KUKA KRL program: EPS_2_25694_SR01_A_20251117072407.src

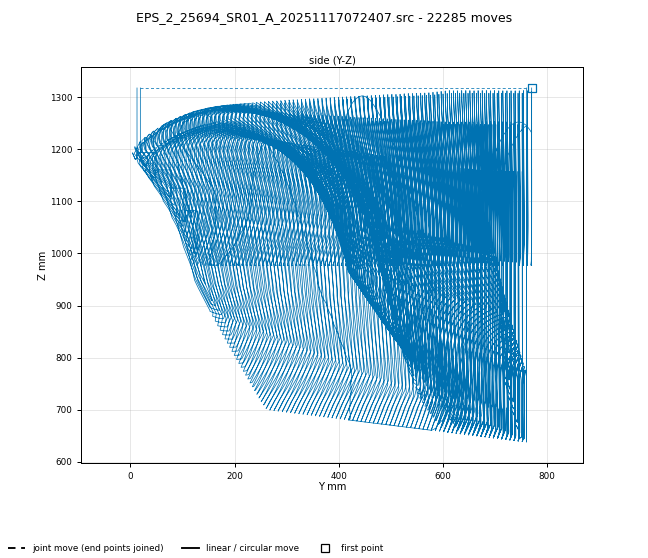
[picture p0: tool path of EPS_2_25694_SR01_A_20251117072407.src, 22285 of 22287 moves have a stored position in this frame; points joined in program order, loops and branches not executed]
&ACCESS RVP
&REL 4
&COMMENT QRS 19112012
&PARAM EDITMASK = *
DEF PART()
EXT BAS (BAS_COMMAND :IN,REAL :IN )
INT I
BAS (#INITMOV,0 )

;KUKA QRS Post kuka4.cps  Date:22-06-2017 !

File_ID=2905

QRS_PRE_INIT()

;Init var - Until changes are made in qrs_pre_init
Outlet_Square_prg=0
Inlet_1_Square_prg=0
Inlet_2_Square_prg=0
Inlet_3_Square_prg=0
Inlet_4_Square_prg=0
Inlet_5_Square_prg=0

Outlet_1={X 0.000, Y 612.000, Z 1041.000, B 0.000, E1 0.000 }
Inlet_1={X 0.000, Y 612.000, Z 981.000, B 0.000, E1 90.000 }
Inlet_2={X 0.000, Y 687.170, Z 452.000, B 0.000, E1 260.000 }
Outlet_1_type=533
Inlet_1_type=533
Inlet_2_type=251
;QRS#1=Sidecore dimensions
;QRS#2=525-21" Concrete
;QRS#3=525-21" Concrete
;QRS#4=250-10" PVC SDR 35
;QRS#5=
;QRS#6=
;QRS#7=
;QRS#8=
;QRS#9=S306-32
;QRS#10=S306-32
;QRS#11=14M PSX
;QRS#12=
;QRS#13=
;QRS#14=
;QRS#15=
;QRS#16=1524x152x1753 5,75'
;QRS#17=EPS Height
;QRS#18=1307,5
;QRS#19=*
;QRS#20= UPDATED VERSION 22-06-2017
;QRS#21=*
Outlet_Square=0350
Inlet_1_Square=0350
Inlet_2_Square=0100
Inlet_3_Square=0
Inlet_4_Square=0
Inlet_5_Square=0
Mill_Square=1
Outlet_Square_Prg=263
Inlet_1_Square_prg=263
Inlet_2_Square_prg=205

QRS_INIT()

$ADVANCE=5

; T1
PTP {E1 171.718,E2 171.718}
PTP {X 0,Y 770.023,A -85,B 0,C 180,E1 171.718,E2 171.718,E3 0,E4 0,E5 0,E6 0}
QRS_SPEED_INIT()
LIN {X 0,Y 770.023,Z 1317.5,A -85,B 0,C 180,E1 171.718,E2 171.718,E3 0,E4 0,E5 0,E6 0} C_VEL
LIN {X 0,Y 770.023,Z 1241.436,A -85,B 0,C 180,E1 171.718,E2 171.718} C_VEL
LIN {X 0,Y 770.023,Z 1233.323,A -85,B 0,C 180,E1 171.718,E2 171.718} C_VEL
LIN {X 0,Y 769.973,Z 1231.44,A -85,B 0,C 180,E1 171.917,E2 171.917} C_VEL
LIN {X 0,Y 769.865,Z 1236.016,A -85,B 0,C 180,E1 172.868,E2 172.868} C_VEL
LIN {X 0,Y 769.858,Z 1240.057,A -85,B 0,C 180,E1 173.85,E2 173.85} C_VEL
LIN {X 0,Y 769.972,Z 1243.895,A -85,B 0,C 180,E1 174.972,E2 174.972} C_VEL
LIN {X 0,Y 769.797,Z 1246.945,A -85,B 0,C 180,E1 176.09,E2 176.09} C_VEL
LIN {X 0,Y 769.867,Z 1249.135,A -85,B 0,C 180,E1 177.209,E2 177.209} C_VEL
LIN {X 0,Y 769.978,Z 1250.214,A -85,B 0,C 180,E1 177.954,E2 177.954} C_VEL
LIN {X 0,Y 769.814,Z 1251.211,A -85,B 0,C 180,E1 179.07,E2 179.07} C_VEL
LIN {X 0,Y 769.987,Z 1251.132,A -85,B 0,C 180,E1 180.93,E2 180.93} C_VEL
LIN {X 0,Y 769.924,Z 1250.495,A -85,B 0,C 180,E1 181.674,E2 181.674} C_VEL
LIN {X 0,Y 769.997,Z 1248.968,A -85,B 0,C 180,E1 182.791,E2 182.791} C_VEL
LIN {X 0,Y 769.853,Z 1246.736,A -85,B 0,C 180,E1 183.909,E2 183.909} C_VEL
LIN {X 0,Y 769.92,Z 1243.606,A -85,B 0,C 180,E1 185.028,E2 185.028} C_VEL
LIN {X 0,Y 769.995,Z 1241.081,A -85,B 0,C 180,E1 185.775,E2 185.775} C_VEL
LIN {X 0,Y 769.852,Z 1237.005,A -85,B 0,C 180,E1 186.824,E2 186.824} C_VEL
LIN {X 0,Y 769.887,Z 1232.516,A -85,B 0,C 180,E1 187.791,E2 187.791} C_VEL
LIN {X 0,Y 769.947,Z 1226.703,A -85,B 0,C 180,E1 188.87,E2 188.87} C_VEL
LIN {X 0,Y 769.873,Z 1220.945,A -85,B 0,C 180,E1 189.814,E2 189.814} C_VEL
LIN {X 0,Y 769.962,Z 1214.413,A -85,B 0,C 180,E1 190.758,E2 190.758} C_VEL
LIN {X 0,Y 769.919,Z 1207.115,A -85,B 0,C 180,E1 191.706,E2 191.706} C_VEL
LIN {X 0,Y 769.869,Z 1200.05,A -85,B 0,C 180,E1 192.54,E2 192.54} C_VEL
LIN {X 0,Y 769.952,Z 1192.23,A -85,B 0,C 180,E1 193.373,E2 193.373} C_VEL
LIN {X 0,Y 769.972,Z 1184.939,A -85,B 0,C 180,E1 194.091,E2 194.091} C_VEL
LIN {X 0,Y 769.933,Z 1175.825,A -85,B 0,C 180,E1 194.91,E2 194.91} C_VEL
LIN {X 0,Y 769.965,Z 1167.286,A -85,B 0,C 180,E1 195.613,E2 195.613} C_VEL
LIN {X 0,Y 769.992,Z 1158.209,A -85,B 0,C 180,E1 196.301,E2 196.301} C_VEL
LIN {X 0,Y 769.94,Z 1148.195,A -85,B 0,C 180,E1 196.999,E2 196.999} C_VEL
LIN {X 0,Y 769.971,Z 1137.702,A -85,B 0,C 180,E1 197.665,E2 197.665} C_VEL
LIN {X 0,Y 769.976,Z 1127.341,A -85,B 0,C 180,E1 198.267,E2 198.267} C_VEL
LIN {X 0,Y 769.983,Z 1116.994,A -85,B 0,C 180,E1 198.819,E2 198.819} C_VEL
LIN {X 0,Y 769.976,Z 1105.571,A -85,B 0,C 180,E1 199.373,E2 199.373} C_VEL
LIN {X 0,Y 769.917,Z 1094.356,A -85,B 0,C 180,E1 199.868,E2 199.868} C_VEL
LIN {X 0,Y 769.976,Z 1080.704,A -85,B 0,C 180,E1 200.4,E2 200.4} C_VEL
LIN {X 0,Y 769.957,Z 1068.91,A -85,B 0,C 180,E1 200.812,E2 200.812} C_VEL
LIN {X 0,Y 769.908,Z 1058.029,A -85,B 0,C 180,E1 201.153,E2 201.153} C_VEL
LIN {X 0,Y 769.994,Z 1042.62,A -85,B 0,C 180,E1 201.561,E2 201.561} C_VEL
LIN {X 0,Y 769.955,Z 1029.278,A -85,B 0,C 180,E1 201.861,E2 201.861} C_VEL
LIN {X 0,Y 769.84,Z 1017.832,A -85,B 0,C 180,E1 202.082,E2 202.082} C_VEL
LIN {X 0,Y 769.939,Z 1002.652,A -85,B 0,C 180,E1 202.304,E2 202.304} C_VEL
LIN {X 0,Y 769.825,Z 984.624,A -85,B 0,C 180,E1 202.504,E2 202.504} C_VEL
LIN {X 0,Y 769.657,Z 979.091,A -85,B 0,C 180,E1 202.564,E2 202.564} C_VEL
LIN {X 0,Y 769.078,Z 977.53,A -85,B 0,C 180,E1 202.604,E2 202.604} C_VEL
LIN {X 0,Y 770.082,Z 977.53,A -85,B 0,C 180,E1 202.974,E2 202.974} C_VEL
LIN {X 0,Y 769.685,Z 977.53,A -85,B 0,C 180,E1 203.948,E2 203.948} C_VEL
LIN {X 0,Y 769.897,Z 977.53,A -85,B 0,C 180,E1 208.082,E2 208.082} C_VEL
LIN {X 0,Y 769.516,Z 977.53,A -85,B 0,C 180,E1 210.601,E2 210.601} C_VEL
LIN {X 0,Y 769.917,Z 977.53,A -85,B 0,C 180,E1 212.388,E2 212.388} C_VEL
LIN {X 0,Y 769.483,Z 977.53,A -85,B 0,C 180,E1 214.641,E2 214.641} C_VEL
LIN {X 0,Y 770.049,Z 977.53,A -85,B 0,C 180,E1 217.324,E2 217.324} C_VEL
LIN {X 0,Y 769.704,Z 977.53,A -85,B 0,C 180,E1 221.735,E2 221.735} C_VEL
LIN {X 0,Y 769.745,Z 977.53,A -85,B 0,C 180,E1 223.064,E2 223.064} C_VEL
LIN {X 0,Y 769.737,Z 977.53,A -85,B 0,C 180,E1 226.937,E2 226.937} C_VEL
LIN {X 0,Y 769.697,Z 977.53,A -85,B 0,C 180,E1 228.264,E2 228.264} C_VEL
LIN {X 0,Y 770.068,Z 977.53,A -85,B 0,C 180,E1 232.674,E2 232.674} C_VEL
LIN {X 0,Y 769.762,Z 977.53,A -85,B 0,C 180,E1 235.892,E2 235.892} C_VEL
LIN {X 0,Y 769.686,Z 977.53,A -85,B 0,C 180,E1 237.601,E2 237.601} C_VEL
LIN {X 0,Y 769.425,Z 977.53,A -85,B 0,C 180,E1 239.767,E2 239.767} C_VEL
LIN {X 0,Y 769.9,Z 977.53,A -85,B 0,C 180,E1 241.918,E2 241.918} C_VEL
LIN {X 0,Y 769.973,Z 977.53,A -85,B 0,C 180,E1 246.365,E2 246.365} C_VEL
LIN {X 0,Y 769.665,Z 977.53,A -85,B 0,C 180,E1 246.705,E2 246.705} C_VEL
LIN {X 0,Y 769.269,Z 977.53,A -85,B 0,C 180,E1 246.754,E2 246.754} C_VEL
LIN {X 0,Y 769.172,Z 977.768,A -85,B 0,C 180,E1 246.767,E2 246.767} C_VEL
LIN {X 0,Y 769.749,Z 993.425,A -85,B 0,C 180,E1 246.941,E2 246.941} C_VEL
LIN {X 0,Y 769.865,Z 1055.898,A -85,B 0,C 180,E1 247.57,E2 247.57} C_VEL
LIN {X 0,Y 769.803,Z 1068.07,A -85,B 0,C 180,E1 247.72,E2 247.72} C_VEL
LIN {X 0,Y 769.924,Z 1081.39,A -85,B 0,C 180,E1 247.941,E2 247.941} C_VEL
LIN {X 0,Y 769.888,Z 1094.597,A -85,B 0,C 180,E1 248.205,E2 248.205} C_VEL
LIN {X 0,Y 769.945,Z 1107.084,A -85,B 0,C 180,E1 248.505,E2 248.505} C_VEL
LIN {X 0,Y 769.959,Z 1120.713,A -85,B 0,C 180,E1 248.887,E2 248.887} C_VEL
LIN {X 0,Y 769.857,Z 1132.612,A -85,B 0,C 180,E1 249.265,E2 249.265} C_VEL
LIN {X 0,Y 769.961,Z 1143.963,A -85,B 0,C 180,E1 249.674,E2 249.674} C_VEL
LIN {X 0,Y 769.976,Z 1156.83,A -85,B 0,C 180,E1 250.195,E2 250.195} C_VEL
LIN {X 0,Y 769.92,Z 1169.12,A -85,B 0,C 180,E1 250.748,E2 250.748} C_VEL
LIN {X 0,Y 769.966,Z 1180.216,A -85,B 0,C 180,E1 251.303,E2 251.303} C_VEL
LIN {X 0,Y 769.976,Z 1191.366,A -85,B 0,C 180,E1 251.915,E2 251.915} C_VEL
LIN {X 0,Y 769.968,Z 1201.997,A -85,B 0,C 180,E1 252.556,E2 252.556} C_VEL
LIN {X 0,Y 769.956,Z 1212.08,A -85,B 0,C 180,E1 253.221,E2 253.221} C_VEL
LIN {X 0,Y 769.966,Z 1221.361,A -85,B 0,C 180,E1 253.887,E2 253.887} C_VEL
LIN {X 0,Y 769.995,Z 1229.576,A -85,B 0,C 180,E1 254.525,E2 254.525} C_VEL
LIN {X 0,Y 769.904,Z 1239.008,A -85,B 0,C 180,E1 255.323,E2 255.323} C_VEL
LIN {X 0,Y 769.901,Z 1246.661,A -85,B 0,C 180,E1 256.027,E2 256.027} C_VEL
LIN {X 0,Y 769.981,Z 1254.955,A -85,B 0,C 180,E1 256.865,E2 256.865} C_VEL
LIN {X 0,Y 769.899,Z 1262.523,A -85,B 0,C 180,E1 257.698,E2 257.698} C_VEL
LIN {X 0,Y 769.889,Z 1269.388,A -85,B 0,C 180,E1 258.53,E2 258.53} C_VEL
LIN {X 0,Y 769.994,Z 1276.399,A -85,B 0,C 180,E1 259.478,E2 259.478} C_VEL
LIN {X 0,Y 769.921,Z 1281.234,A -85,B 0,C 180,E1 260.186,E2 260.186} C_VEL
LIN {X 0,Y 769.846,Z 1286.993,A -85,B 0,C 180,E1 261.128,E2 261.128} C_VEL
LIN {X 0,Y 769.955,Z 1292.809,A -85,B 0,C 180,E1 262.232,E2 262.232} C_VEL
LIN {X 0,Y 769.885,Z 1297.298,A -85,B 0,C 180,E1 263.207,E2 263.207} C_VEL
LIN {X 0,Y 769.849,Z 1301.265,A -85,B 0,C 180,E1 264.223,E2 264.223} C_VEL
LIN {X 0,Y 769.951,Z 1303.746,A -85,B 0,C 180,E1 264.971,E2 264.971} C_VEL
LIN {X 0,Y 769.854,Z 1306.835,A -85,B 0,C 180,E1 266.09,E2 266.09} C_VEL
LIN {X 0,Y 769.819,Z 1309.08,A -85,B 0,C 180,E1 267.207,E2 267.207} C_VEL
LIN {X 0,Y 769.983,Z 1310.517,A -85,B 0,C 180,E1 268.325,E2 268.325} C_VEL
LIN {X 0,Y 769.856,Z 1311.187,A -85,B 0,C 180,E1 269.069,E2 269.069} C_VEL
LIN {X 0,Y 769.856,Z 1311.188,A -85,B 0,C 180,E1 270.929,E2 270.929} C_VEL
LIN {X 0,Y 769.923,Z 1310.164,A -85,B 0,C 180,E1 272.045,E2 272.045} C_VEL
LIN {X 0,Y 769.819,Z 1309.084,A -85,B 0,C 180,E1 272.79,E2 272.79} C_VEL
LIN {X 0,Y 769.853,Z 1306.84,A -85,B 0,C 180,E1 273.908,E2 273.908} C_VEL
LIN {X 0,Y 769.952,Z 1303.754,A -85,B 0,C 180,E1 275.027,E2 275.027} C_VEL
LIN {X 0,Y 769.844,Z 1299.884,A -85,B 0,C 180,E1 276.149,E2 276.149} C_VEL
LIN {X 0,Y 769.925,Z 1295.884,A -85,B 0,C 180,E1 277.111,E2 277.111} C_VEL
LIN {X 0,Y 769.924,Z 1291.346,A -85,B 0,C 180,E1 278.059,E2 278.059} C_VEL
LIN {X 0,Y 769.846,Z 1287.007,A -85,B 0,C 180,E1 278.87,E2 278.87} C_VEL
LIN {X 0,Y 769.921,Z 1281.25,A -85,B 0,C 180,E1 279.812,E2 279.812} C_VEL
LIN {X 0,Y 769.972,Z 1274.763,A -85,B 0,C 180,E1 280.756,E2 280.756} C_VEL
LIN {X 0,Y 769.879,Z 1267.512,A -85,B 0,C 180,E1 281.706,E2 281.706} C_VEL
LIN {X 0,Y 769.935,Z 1260.465,A -85,B 0,C 180,E1 282.537,E2 282.537} C_VEL
LIN {X 0,Y 769.965,Z 1252.697,A -85,B 0,C 180,E1 283.371,E2 283.371} C_VEL
LIN {X 0,Y 769.895,Z 1243.731,A -85,B 0,C 180,E1 284.248,E2 284.248} C_VEL
LIN {X 0,Y 769.951,Z 1236.134,A -85,B 0,C 180,E1 284.929,E2 284.929} C_VEL
LIN {X 0,Y 769.974,Z 1226.492,A -85,B 0,C 180,E1 285.719,E2 285.719} C_VEL
LIN {X 0,Y 769.941,Z 1217.541,A -85,B 0,C 180,E1 286.395,E2 286.395} C_VEL
LIN {X 0,Y 769.96,Z 1207.794,A -85,B 0,C 180,E1 287.069,E2 287.069} C_VEL
LIN {X 0,Y 769.966,Z 1198.499,A -85,B 0,C 180,E1 287.663,E2 287.663} C_VEL
LIN {X 0,Y 769.97,Z 1187.07,A -85,B 0,C 180,E1 288.327,E2 288.327} C_VEL
LIN {X 0,Y 769.963,Z 1176.692,A -85,B 0,C 180,E1 288.879,E2 288.879} C_VEL
LIN {X 0,Y 769.934,Z 1165.232,A -85,B 0,C 180,E1 289.434,E2 289.434} C_VEL
LIN {X 0,Y 769.98,Z 1153.974,A -85,B 0,C 180,E1 289.926,E2 289.926} C_VEL
LIN {X 0,Y 769.953,Z 1140.728,A -85,B 0,C 180,E1 290.445,E2 290.445} C_VEL
LIN {X 0,Y 769.903,Z 1129.904,A -85,B 0,C 180,E1 290.827,E2 290.827} C_VEL
LIN {X 0,Y 769.98,Z 1116.504,A -85,B 0,C 180,E1 291.238,E2 291.238} C_VEL
LIN {X 0,Y 769.907,Z 1102.481,A -85,B 0,C 180,E1 291.612,E2 291.612} C_VEL
LIN {X 0,Y 769.923,Z 1090.854,A -85,B 0,C 180,E1 291.877,E2 291.877} C_VEL
LIN {X 0,Y 769.91,Z 1076.317,A -85,B 0,C 180,E1 292.149,E2 292.149} C_VEL
LIN {X 0,Y 769.82,Z 1064.258,A -85,B 0,C 180,E1 292.334,E2 292.334} C_VEL
LIN {X 0,Y 769.844,Z 1045.508,A -85,B 0,C 180,E1 292.54,E2 292.54} C_VEL
LIN {X 0,Y 769.588,Z 1005.253,A -85,B 0,C 180,E1 292.947,E2 292.947} C_VEL
LIN {X 0,Y 769.15,Z 977.543,A -85,B 0,C 180,E1 293.236,E2 293.236} C_VEL
LIN {X 0,Y 769.593,Z 977.53,A -85,B 0,C 180,E1 293.285,E2 293.285} C_VEL
LIN {X 0,Y 769.974,Z 977.53,A -85,B 0,C 180,E1 293.624,E2 293.624} C_VEL
LIN {X 0,Y 769.901,Z 977.53,A -85,B 0,C 180,E1 298.08,E2 298.08} C_VEL
LIN {X 0,Y 769.513,Z 977.53,A -85,B 0,C 180,E1 300.601,E2 300.601} C_VEL
LIN {X 0,Y 769.891,Z 977.53,A -85,B 0,C 180,E1 302.387,E2 302.387} C_VEL
LIN {X 0,Y 769.475,Z 977.53,A -85,B 0,C 180,E1 304.639,E2 304.639} C_VEL
LIN {X 0,Y 770.07,Z 977.53,A -85,B 0,C 180,E1 307.326,E2 307.326} C_VEL
LIN {X 0,Y 769.805,Z 977.53,A -85,B 0,C 180,E1 311.726,E2 311.726} C_VEL
LIN {X 0,Y 769.853,Z 977.53,A -85,B 0,C 180,E1 313.073,E2 313.073} C_VEL
LIN {X 0,Y 769.844,Z 977.53,A -85,B 0,C 180,E1 314.267,E2 314.267} C_VEL
LIN {X 0,Y 769.751,Z 977.53,A -85,B 0,C 180,E1 315.724,E2 315.724} C_VEL
LIN {X 0,Y 769.775,Z 977.53,A -85,B 0,C 180,E1 319.729,E2 319.729} C_VEL
LIN {X 0,Y 769.825,Z 977.53,A -85,B 0,C 180,E1 320.72,E2 320.72} C_VEL
LIN {X 0,Y 769.434,Z 977.53,A -85,B 0,C 180,E1 323.062,E2 323.062} C_VEL
LIN {X 0,Y 769.866,Z 977.53,A -85,B 0,C 180,E1 325.379,E2 325.379} C_VEL
LIN {X 0,Y 770.006,Z 977.53,A -85,B 0,C 180,E1 329.333,E2 329.333} C_VEL
LIN {X 0,Y 769.849,Z 977.53,A -85,B 0,C 180,E1 333.226,E2 333.226} C_VEL
LIN {X 0,Y 769.942,Z 977.53,A -85,B 0,C 180,E1 334.008,E2 334.008} C_VEL
LIN {X 0,Y 770.006,Z 977.53,A -85,B 0,C 180,E1 337.678,E2 337.678} C_VEL
LIN {X 0,Y 769.978,Z 977.53,A -85,B 0,C 180,E1 338.081,E2 338.081} C_VEL
LIN {X 0,Y 770,Z 977.53,A -85,B 0,C 180,E1 342.039,E2 342.039} C_VEL
LIN {X 0,Y 769.718,Z 977.53,A -85,B 0,C 180,E1 343.978,E2 343.978} C_VEL
LIN {X 0,Y 769.807,Z 977.53,A -85,B 0,C 180,E1 345.906,E2 345.906} C_VEL
LIN {X 0,Y 770.015,Z 977.53,A -85,B 0,C 180,E1 349.716,E2 349.716} C_VEL
LIN {X 0,Y 770.022,Z 977.53,A -85,B 0,C 180,E1 353.477,E2 353.477} C_VEL
LIN {X 0,Y 770.079,Z 977.53,A -85,B 0,C 180,E1 357.209,E2 357.209} C_VEL
LIN {X 0,Y 769.87,Z 977.53,A -85,B 0,C 180,E1 357.945,E2 357.945} C_VEL
LIN {X 0,Y 770.003,Z 1029.792,A -85,B 0,C 180,E1 358.443,E2 358.443} C_VEL
LIN {X 0,Y 770.057,Z 1040.253,A -85,B 0,C 180,E1 358.589,E2 358.589} C_VEL
LIN {X 0,Y 770.026,Z 1050.198,A -85,B 0,C 180,E1 358.784,E2 358.784} C_VEL
LIN {X 0,Y 770.011,Z 1058.48,A -85,B 0,C 180,E1 358.985,E2 358.985} C_VEL
LIN {X 0,Y 770.028,Z 1067.655,A -85,B 0,C 180,E1 359.256,E2 359.256} C_VEL
LIN {X 0,Y 769.994,Z 1075.609,A -85,B 0,C 180,E1 359.535,E2 359.535} C_VEL
LIN {X 0,Y 770.029,Z 1083.642,A -85,B 0,C 180,E1 359.861,E2 359.861} C_VEL
LIN {X 0,Y 770.033,Z 1092.613,A -85,B 0,C 180,E1 360.279,E2 360.279} C_VEL
LIN {X 0,Y 770.022,Z 1099.542,A -85,B 0,C 180,E1 360.651,E2 360.651} C_VEL
LIN {X 0,Y 770.027,Z 1105.762,A -85,B 0,C 180,E1 361.023,E2 361.023} C_VEL
LIN {X 0,Y 770.025,Z 1112.753,A -85,B 0,C 180,E1 361.488,E2 361.488} C_VEL
LIN {X 0,Y 770.007,Z 1123.426,A -85,B 0,C 180,E1 362.325,E2 362.325} C_VEL
LIN {X 0,Y 769.995,Z 1128.51,A -85,B 0,C 180,E1 362.791,E2 362.791} C_VEL
LIN {X 0,Y 769.999,Z 1133.968,A -85,B 0,C 180,E1 363.35,E2 363.35} C_VEL
LIN {X 0,Y 770.012,Z 1138.814,A -85,B 0,C 180,E1 363.909,E2 363.909} C_VEL
LIN {X 0,Y 769.97,Z 1144.348,A -85,B 0,C 180,E1 364.655,E2 364.655} C_VEL
LIN {X 0,Y 770.009,Z 1149.025,A -85,B 0,C 180,E1 365.401,E2 365.401} C_VEL
LIN {X 0,Y 769.985,Z 1152.84,A -85,B 0,C 180,E1 366.149,E2 366.149} C_VEL
LIN {X 0,Y 769.947,Z 1155.711,A -85,B 0,C 180,E1 366.829,E2 366.829} C_VEL
LIN {X 0,Y 769.992,Z 1157.731,A -85,B 0,C 180,E1 367.438,E2 367.438} C_VEL
LIN {X 0,Y 769.973,Z 1160.024,A -85,B 0,C 180,E1 368.4,E2 368.4} C_VEL
LIN {X 0,Y 769.979,Z 1161.182,A -85,B 0,C 180,E1 369.341,E2 369.341} C_VEL
LIN {X 0,Y 769.995,Z 1161.379,A -85,B 0,C 180,E1 369.812,E2 369.812} C_VEL
LIN {X 0,Y 769.982,Z 1161.328,A -85,B 0,C 180,E1 370.284,E2 370.284} C_VEL
LIN {X 0,Y 769.956,Z 1161.022,A -85,B 0,C 180,E1 370.758,E2 370.758} C_VEL
LIN {X 0,Y 769.955,Z 1160.453,A -85,B 0,C 180,E1 371.231,E2 371.231} C_VEL
LIN {X 0,Y 769.981,Z 1159.617,A -85,B 0,C 180,E1 371.705,E2 371.705} C_VEL
LIN {X 0,Y 770.005,Z 1158.515,A -85,B 0,C 180,E1 372.18,E2 372.18} C_VEL
LIN {X 0,Y 769.974,Z 1157.15,A -85,B 0,C 180,E1 372.657,E2 372.657} C_VEL
LIN {X 0,Y 769.949,Z 1154.542,A -85,B 0,C 180,E1 373.373,E2 373.373} C_VEL
LIN {X 0,Y 770.009,Z 1151.27,A -85,B 0,C 180,E1 374.09,E2 374.09} C_VEL
LIN {X 0,Y 770.001,Z 1148.916,A -85,B 0,C 180,E1 374.529,E2 374.529} C_VEL
LIN {X 0,Y 769.965,Z 1144.543,A -85,B 0,C 180,E1 375.227,E2 375.227} C_VEL
LIN {X 0,Y 769.982,Z 1140.244,A -85,B 0,C 180,E1 375.819,E2 375.819} C_VEL
LIN {X 0,Y 770.008,Z 1135.406,A -85,B 0,C 180,E1 376.404,E2 376.404} C_VEL
LIN {X 0,Y 769.984,Z 1130.358,A -85,B 0,C 180,E1 376.939,E2 376.939} C_VEL
LIN {X 0,Y 769.995,Z 1125.764,A -85,B 0,C 180,E1 377.376,E2 377.376} C_VEL
LIN {X 0,Y 769.985,Z 1120.622,A -85,B 0,C 180,E1 377.815,E2 377.815} C_VEL
LIN {X 0,Y 770.008,Z 1112.349,A -85,B 0,C 180,E1 378.45,E2 378.45} C_VEL
LIN {X 0,Y 770.01,Z 1104.911,A -85,B 0,C 180,E1 378.941,E2 378.941} C_VEL
LIN {X 0,Y 769.994,Z 1096.412,A -85,B 0,C 180,E1 379.434,E2 379.434} C_VEL
LIN {X 0,Y 770.023,Z 1089.066,A -85,B 0,C 180,E1 379.803,E2 379.803} C_VEL
LIN {X 0,Y 770.024,Z 1079.515,A -85,B 0,C 180,E1 380.225,E2 380.225} C_VEL
LIN {X 0,Y 770.003,Z 1071.513,A -85,B 0,C 180,E1 380.524,E2 380.524} C_VEL
LIN {X 0,Y 770.047,Z 1063.09,A -85,B 0,C 180,E1 380.793,E2 380.793} C_VEL
LIN {X 0,Y 770.012,Z 1053.214,A -85,B 0,C 180,E1 381.06,E2 381.06} C_VEL
LIN {X 0,Y 770.017,Z 1043.273,A -85,B 0,C 180,E1 381.266,E2 381.266} C_VEL
LIN {X 0,Y 769.958,Z 1033.431,A -85,B 0,C 180,E1 381.425,E2 381.425} C_VEL
LIN {X 0,Y 769.977,Z 1018.248,A -85,B 0,C 180,E1 381.581,E2 381.581} C_VEL
LIN {X 0,Y 769.862,Z 988.278,A -85,B 0,C 180,E1 381.864,E2 381.864} C_VEL
LIN {X 0,Y 769.329,Z 977.53,A -85,B 0,C 180,E1 381.98,E2 381.98} C_VEL
LIN {X 0,Y 769.736,Z 977.53,A -85,B 0,C 180,E1 382.036,E2 382.036} C_VEL
LIN {X 0,Y 770.051,Z 977.53,A -85,B 0,C 180,E1 382.135,E2 382.135} C_VEL
LIN {X 0,Y 770,Z 977.53,A -85,B 0,C 180,E1 383.938,E2 383.938} C_VEL
LIN {X 0,Y 769.573,Z 977.53,A -85,B 0,C 180,E1 386.734,E2 386.734} C_VEL
LIN {X 0,Y 769.923,Z 977.53,A -85,B 0,C 180,E1 388.081,E2 388.081} C_VEL
LIN {X 0,Y 769.527,Z 977.53,A -85,B 0,C 180,E1 390.607,E2 390.607} C_VEL
LIN {X 0,Y 769.91,Z 977.53,A -85,B 0,C 180,E1 392.388,E2 392.388} C_VEL
LIN {X 0,Y 769.477,Z 977.53,A -85,B 0,C 180,E1 394.641,E2 394.641} C_VEL
LIN {X 0,Y 770.051,Z 977.53,A -85,B 0,C 180,E1 397.328,E2 397.328} C_VEL
LIN {X 0,Y 769.806,Z 977.53,A -85,B 0,C 180,E1 401.728,E2 401.728} C_VEL
LIN {X 0,Y 769.865,Z 977.53,A -85,B 0,C 180,E1 403.076,E2 403.076} C_VEL
LIN {X 0,Y 769.853,Z 977.53,A -85,B 0,C 180,E1 404.269,E2 404.269} C_VEL
LIN {X 0,Y 769.769,Z 977.53,A -85,B 0,C 180,E1 405.728,E2 405.728} C_VEL
LIN {X 0,Y 769.807,Z 977.53,A -85,B 0,C 180,E1 409.729,E2 409.729} C_VEL
LIN {X 0,Y 769.846,Z 977.53,A -85,B 0,C 180,E1 410.723,E2 410.723} C_VEL
LIN {X 0,Y 769.447,Z 977.53,A -85,B 0,C 180,E1 413.065,E2 413.065} C_VEL
LIN {X 0,Y 769.869,Z 977.53,A -85,B 0,C 180,E1 415.381,E2 415.381} C_VEL
LIN {X 0,Y 770.013,Z 977.53,A -85,B 0,C 180,E1 419.336,E2 419.336} C_VEL
LIN {X 0,Y 769.846,Z 977.53,A -85,B 0,C 180,E1 423.231,E2 423.231} C_VEL
LIN {X 0,Y 769.94,Z 977.53,A -85,B 0,C 180,E1 424.01,E2 424.01} C_VEL
LIN {X 0,Y 770.005,Z 977.53,A -85,B 0,C 180,E1 427.684,E2 427.684} C_VEL
LIN {X 0,Y 769.974,Z 977.53,A -85,B 0,C 180,E1 428.082,E2 428.082} C_VEL
LIN {X 0,Y 769.984,Z 977.53,A -85,B 0,C 180,E1 432.04,E2 432.04} C_VEL
LIN {X 0,Y 769.723,Z 977.53,A -85,B 0,C 180,E1 433.979,E2 433.979} C_VEL
LIN {X 0,Y 769.825,Z 977.53,A -85,B 0,C 180,E1 435.908,E2 435.908} C_VEL
LIN {X 0,Y 770.041,Z 977.53,A -85,B 0,C 180,E1 439.718,E2 439.718} C_VEL
LIN {X 0,Y 770.051,Z 977.53,A -85,B 0,C 180,E1 443.478,E2 443.478} C_VEL
LIN {X 0,Y 770.057,Z 977.53,A -85,B 0,C 180,E1 447.211,E2 447.211} C_VEL
LIN {X 0,Y 770.073,Z 977.53,A -85,B 0,C 180,E1 450.931,E2 450.931} C_VEL
LIN {X 0,Y 770.044,Z 977.53,A -85,B 0,C 180,E1 454.655,E2 454.655} C_VEL
LIN {X 0,Y 770.025,Z 977.53,A -85,B 0,C 180,E1 458.4,E2 458.4} C_VEL
LIN {X 0,Y 770.008,Z 977.53,A -85,B 0,C 180,E1 462.181,E2 462.181} C_VEL
LIN {X 0,Y 769.993,Z 977.53,A -85,B 0,C 180,E1 466.017,E2 466.017} C_VEL
LIN {X 0,Y 769.867,Z 977.53,A -85,B 0,C 180,E1 466.718,E2 466.718} C_VEL
LIN {X 0,Y 769.984,Z 977.53,A -85,B 0,C 180,E1 469.929,E2 469.929} C_VEL
LIN {X 0,Y 769.592,Z 977.53,A -85,B 0,C 180,E1 472.241,E2 472.241} C_VEL
LIN {X 0,Y 769.949,Z 977.53,A -85,B 0,C 180,E1 473.941,E2 473.941} C_VEL
LIN {X 0,Y 769.578,Z 977.53,A -85,B 0,C 180,E1 476.73,E2 476.73} C_VEL
LIN {X 0,Y 769.921,Z 977.53,A -85,B 0,C 180,E1 478.082,E2 478.082} C_VEL
LIN {X 0,Y 769.515,Z 977.53,A -85,B 0,C 180,E1 480.601,E2 480.601} C_VEL
LIN {X 0,Y 769.885,Z 977.53,A -85,B 0,C 180,E1 482.39,E2 482.39} C_VEL
LIN {X 0,Y 769.563,Z 977.53,A -85,B 0,C 180,E1 484.086,E2 484.086} C_VEL
LIN {X 0,Y 770.068,Z 977.53,A -85,B 0,C 180,E1 487.326,E2 487.326} C_VEL
LIN {X 0,Y 769.797,Z 977.53,A -85,B 0,C 180,E1 491.729,E2 491.729} C_VEL
LIN {X 0,Y 769.864,Z 977.53,A -85,B 0,C 180,E1 493.074,E2 493.074} C_VEL
LIN {X 0,Y 769.852,Z 977.53,A -85,B 0,C 180,E1 494.269,E2 494.269} C_VEL
LIN {X 0,Y 769.778,Z 977.53,A -85,B 0,C 180,E1 495.726,E2 495.726} C_VEL
LIN {X 0,Y 769.809,Z 977.53,A -85,B 0,C 180,E1 499.73,E2 499.73} C_VEL
LIN {X 0,Y 769.841,Z 977.53,A -85,B 0,C 180,E1 500.721,E2 500.721} C_VEL
LIN {X 0,Y 769.435,Z 977.53,A -85,B 0,C 180,E1 503.062,E2 503.062} C_VEL
LIN {X 0,Y 769.87,Z 977.53,A -85,B 0,C 180,E1 505.379,E2 505.379} C_VEL
LIN {X 0,Y 770.015,Z 977.53,A -85,B 0,C 180,E1 509.336,E2 509.336} C_VEL
LIN {X 0,Y 769.856,Z 977.53,A -85,B 0,C 180,E1 513.23,E2 513.23} C_VEL
LIN {X 0,Y 769.974,Z 977.53,A -85,B 0,C 180,E1 514.009,E2 514.009} C_VEL
LIN {X 0,Y 770.006,Z 977.53,A -85,B 0,C 180,E1 517.136,E2 517.136} C_VEL
LIN {X 0,Y 769.397,Z 977.53,A -85,B 0,C 180,E1 517.252,E2 517.252} C_VEL
LIN {X 0,Y 768.845,Z 977.53,A -85,B 0,C 180,E1 517.305,E2 517.305} C_VEL
LIN {X 0,Y 769.772,Z 988.712,A -85,B 0,C 180,E1 517.444,E2 517.444} C_VEL
LIN {X 0,Y 769.823,Z 1007.209,A -85,B 0,C 180,E1 517.663,E2 517.663} C_VEL
LIN {X 0,Y 769.975,Z 1021.434,A -85,B 0,C 180,E1 517.898,E2 517.898} C_VEL
LIN {X 0,Y 770.014,Z 1034.601,A -85,B 0,C 180,E1 518.164,E2 518.164} C_VEL
LIN {X 0,Y 769.952,Z 1046.898,A -85,B 0,C 180,E1 518.455,E2 518.455} C_VEL
LIN {X 0,Y 769.92,Z 1057.218,A -85,B 0,C 180,E1 518.734,E2 518.734} C_VEL
LIN {X 0,Y 769.964,Z 1072.044,A -85,B 0,C 180,E1 519.203,E2 519.203} C_VEL
LIN {X 0,Y 769.908,Z 1085.143,A -85,B 0,C 180,E1 519.675,E2 519.675} C_VEL
LIN {X 0,Y 769.974,Z 1096.471,A -85,B 0,C 180,E1 520.134,E2 520.134} C_VEL
LIN {X 0,Y 769.984,Z 1108.8,A -85,B 0,C 180,E1 520.689,E2 520.689} C_VEL
LIN {X 0,Y 769.948,Z 1119.93,A -85,B 0,C 180,E1 521.242,E2 521.242} C_VEL
LIN {X 0,Y 769.965,Z 1131.109,A -85,B 0,C 180,E1 521.855,E2 521.855} C_VEL
LIN {X 0,Y 769.978,Z 1141.42,A -85,B 0,C 180,E1 522.474,E2 522.474} C_VEL
LIN {X 0,Y 769.987,Z 1151.359,A -85,B 0,C 180,E1 523.126,E2 523.126} C_VEL
LIN {X 0,Y 769.953,Z 1160.642,A -85,B 0,C 180,E1 523.786,E2 523.786} C_VEL
LIN {X 0,Y 769.952,Z 1170.522,A -85,B 0,C 180,E1 524.558,E2 524.558} C_VEL
LIN {X 0,Y 769.997,Z 1178.48,A -85,B 0,C 180,E1 525.233,E2 525.233} C_VEL
LIN {X 0,Y 769.985,Z 1187.109,A -85,B 0,C 180,E1 526.029,E2 526.029} C_VEL
LIN {X 0,Y 769.958,Z 1195.381,A -85,B 0,C 180,E1 526.866,E2 526.866} C_VEL
LIN {X 0,Y 769.885,Z 1202.908,A -85,B 0,C 180,E1 527.699,E2 527.699} C_VEL
LIN {X 0,Y 769.93,Z 1209.726,A -85,B 0,C 180,E1 528.531,E2 528.531} C_VEL
LIN {X 0,Y 769.992,Z 1215.088,A -85,B 0,C 180,E1 529.243,E2 529.243} C_VEL
LIN {X 0,Y 769.861,Z 1221.549,A -85,B 0,C 180,E1 530.186,E2 530.186} C_VEL
LIN {X 0,Y 769.865,Z 1227.254,A -85,B 0,C 180,E1 531.129,E2 531.129} C_VEL
LIN {X 0,Y 769.973,Z 1231.44,A -85,B 0,C 180,E1 531.917,E2 531.917} C_VEL
LIN {X 0,Y 765.947,Z 1237.912,A -85,B 0,C 180,E1 533.106,E2 533.106} C_VEL
LIN {X 0,Y 762.08,Z 1242.862,A -85,B 0,C 180,E1 534.327,E2 534.327} C_VEL
LIN {X 0,Y 761.989,Z 1249.004,A -85,B 0,C 180,E1 536.572,E2 536.572} C_VEL
LIN {X 0,Y 762.019,Z 1252.113,A -85,B 0,C 180,E1 538.853,E2 538.853} C_VEL
LIN {X 0,Y 762.149,Z 1252.048,A -85,B 0,C 180,E1 541.131,E2 541.131} C_VEL
LIN {X 0,Y 762.035,Z 1247.623,A -85,B 0,C 180,E1 543.982,E2 543.982} C_VEL
LIN {X 0,Y 762.057,Z 1238.049,A -85,B 0,C 180,E1 546.843,E2 546.843} C_VEL
LIN {X 0,Y 762.086,Z 1222.822,A -85,B 0,C 180,E1 549.721,E2 549.721} C_VEL
LIN {X 0,Y 762.11,Z 1200.866,A -85,B 0,C 180,E1 552.623,E2 552.623} C_VEL
LIN {X 0,Y 762.202,Z 1175.44,A -85,B 0,C 180,E1 555.115,E2 555.115} C_VEL
LIN {X 0,Y 762.269,Z 1145.776,A -85,B 0,C 180,E1 557.337,E2 557.337} C_VEL
LIN {X 0,Y 762.415,Z 1113.078,A -85,B 0,C 180,E1 559.208,E2 559.208} C_VEL
LIN {X 0,Y 762.52,Z 1077.64,A -85,B 0,C 180,E1 560.719,E2 560.719} C_VEL
LIN {X 0,Y 762.64,Z 1040.827,A -85,B 0,C 180,E1 561.822,E2 561.822} C_VEL
LIN {X 0,Y 762.66,Z 1003.996,A -85,B 0,C 180,E1 562.513,E2 562.513} C_VEL
LIN {X 0,Y 761.71,Z 977.53,A -85,B 0,C 180,E1 562.852,E2 562.852} C_VEL
LIN {X 0,Y 761.713,Z 977.53,A -85,B 0,C 180,E1 568.932,E2 568.932} C_VEL
LIN {X 0,Y 761.71,Z 977.53,A -85,B 0,C 180,E1 573.342,E2 573.342} C_VEL
LIN {X 0,Y 761.804,Z 977.53,A -85,B 0,C 180,E1 578.053,E2 578.053} C_VEL
LIN {X 0,Y 761.813,Z 977.53,A -85,B 0,C 180,E1 582.621,E2 582.621} C_VEL
LIN {X 0,Y 761.791,Z 977.53,A -85,B 0,C 180,E1 587.453,E2 587.453} C_VEL
LIN {X 0,Y 761.919,Z 977.53,A -85,B 0,C 180,E1 593.378,E2 593.378} C_VEL
LIN {X 0,Y 761.785,Z 977.53,A -85,B 0,C 180,E1 597.523,E2 597.523} C_VEL
LIN {X 0,Y 761.652,Z 977.53,A -85,B 0,C 180,E1 602.775,E2 602.775} C_VEL
LIN {X 0,Y 761.911,Z 978.328,A -85,B 0,C 180,E1 606.538,E2 606.538} C_VEL
LIN {X 0,Y 762.567,Z 1074.232,A -85,B 0,C 180,E1 607.594,E2 607.594} C_VEL
LIN {X 0,Y 762.569,Z 1112.633,A -85,B 0,C 180,E1 608.438,E2 608.438} C_VEL
LIN {X 0,Y 762.46,Z 1148.647,A -85,B 0,C 180,E1 609.654,E2 609.654} C_VEL
LIN {X 0,Y 762.355,Z 1183.951,A -85,B 0,C 180,E1 611.312,E2 611.312} C_VEL
LIN {X 0,Y 762.251,Z 1216.126,A -85,B 0,C 180,E1 613.327,E2 613.327} C_VEL
LIN {X 0,Y 762.164,Z 1245.722,A -85,B 0,C 180,E1 615.763,E2 615.763} C_VEL
LIN {X 0,Y 762.087,Z 1269.751,A -85,B 0,C 180,E1 618.391,E2 618.391} C_VEL
LIN {X 0,Y 762.027,Z 1288.279,A -85,B 0,C 180,E1 621.14,E2 621.14} C_VEL
LIN {X 0,Y 762.033,Z 1301.544,A -85,B 0,C 180,E1 623.986,E2 623.986} C_VEL
LIN {X 0,Y 761.996,Z 1308.937,A -85,B 0,C 180,E1 626.585,E2 626.585} C_VEL
LIN {X 0,Y 762.068,Z 1312.085,A -85,B 0,C 180,E1 628.866,E2 628.866} C_VEL
LIN {X 0,Y 762.037,Z 1312.076,A -85,B 0,C 180,E1 631.145,E2 631.145} C_VEL
LIN {X 0,Y 762.056,Z 1307.704,A -85,B 0,C 180,E1 633.996,E2 633.996} C_VEL
LIN {X 0,Y 762.108,Z 1296.903,A -85,B 0,C 180,E1 637.144,E2 637.144} C_VEL
LIN {X 0,Y 762.111,Z 1281.123,A -85,B 0,C 180,E1 640.024,E2 640.024} C_VEL
LIN {X 0,Y 762.173,Z 1260.035,A -85,B 0,C 180,E1 642.758,E2 642.758} C_VEL
LIN {X 0,Y 762.218,Z 1234.031,A -85,B 0,C 180,E1 645.278,E2 645.278} C_VEL
LIN {X 0,Y 762.307,Z 1204.374,A -85,B 0,C 180,E1 647.473,E2 647.473} C_VEL
LIN {X 0,Y 762.401,Z 1170.617,A -85,B 0,C 180,E1 649.375,E2 649.375} C_VEL
LIN {X 0,Y 762.462,Z 1133.124,A -85,B 0,C 180,E1 650.928,E2 650.928} C_VEL
LIN {X 0,Y 762.592,Z 1092.164,A -85,B 0,C 180,E1 652.071,E2 652.071} C_VEL
LIN {X 0,Y 762.592,Z 1053.334,A -85,B 0,C 180,E1 652.687,E2 652.687} C_VEL
LIN {X 0,Y 761.925,Z 977.53,A -85,B 0,C 180,E1 653.498,E2 653.498} C_VEL
LIN {X 0,Y 761.718,Z 977.53,A -85,B 0,C 180,E1 658.951,E2 658.951} C_VEL
LIN {X 0,Y 761.667,Z 977.53,A -85,B 0,C 180,E1 663.352,E2 663.352} C_VEL
LIN {X 0,Y 761.801,Z 977.53,A -85,B 0,C 180,E1 668.075,E2 668.075} C_VEL
LIN {X 0,Y 761.916,Z 977.53,A -85,B 0,C 180,E1 672.641,E2 672.641} C_VEL
LIN {X 0,Y 761.783,Z 977.53,A -85,B 0,C 180,E1 675.896,E2 675.896} C_VEL
LIN {X 0,Y 761.872,Z 977.53,A -85,B 0,C 180,E1 680.873,E2 680.873} C_VEL
LIN {X 0,Y 761.702,Z 977.53,A -85,B 0,C 180,E1 686.165,E2 686.165} C_VEL
LIN {X 0,Y 761.783,Z 977.53,A -85,B 0,C 180,E1 690.193,E2 690.193} C_VEL
LIN {X 0,Y 762.015,Z 977.53,A -85,B 0,C 180,E1 694.07,E2 694.07} C_VEL
LIN {X 0,Y 762.123,Z 977.53,A -85,B 0,C 180,E1 697.817,E2 697.817} C_VEL
LIN {X 0,Y 761.907,Z 977.53,A -85,B 0,C 180,E1 702.689,E2 702.689} C_VEL
LIN {X 0,Y 761.585,Z 977.53,A -85,B 0,C 180,E1 707.368,E2 707.368} C_VEL
LIN {X 0,Y 761.778,Z 977.53,A -85,B 0,C 180,E1 710.853,E2 710.853} C_VEL
LIN {X 0,Y 761.853,Z 977.53,A -85,B 0,C 180,E1 714.302,E2 714.302} C_VEL
LIN {X 0,Y 762,Z 977.53,A -85,B 0,C 180,E1 717.8,E2 717.8} C_VEL
LIN {X 0,Y 762.363,Z 1043.05,A -85,B 0,C 180,E1 718.513,E2 718.513} C_VEL
LIN {X 0,Y 762.297,Z 1071.501,A -85,B 0,C 180,E1 719.261,E2 719.261} C_VEL
LIN {X 0,Y 762.284,Z 1098.022,A -85,B 0,C 180,E1 720.435,E2 720.435} C_VEL
LIN {X 0,Y 762.239,Z 1121.159,A -85,B 0,C 180,E1 722.002,E2 722.002} C_VEL
LIN {X 0,Y 762.213,Z 1139.734,A -85,B 0,C 180,E1 723.855,E2 723.855} C_VEL
LIN {X 0,Y 762.178,Z 1153.148,A -85,B 0,C 180,E1 725.965,E2 725.965} C_VEL
LIN {X 0,Y 762.146,Z 1160.305,A -85,B 0,C 180,E1 728.007,E2 728.007} C_VEL
LIN {X 0,Y 762.164,Z 1162.401,A -85,B 0,C 180,E1 730.314,E2 730.314} C_VEL
LIN {X 0,Y 762.191,Z 1159.967,A -85,B 0,C 180,E1 732.056,E2 732.056} C_VEL
LIN {X 0,Y 762.187,Z 1152.402,A -85,B 0,C 180,E1 734.102,E2 734.102} C_VEL
LIN {X 0,Y 762.183,Z 1138.795,A -85,B 0,C 180,E1 736.167,E2 736.167} C_VEL
LIN {X 0,Y 762.188,Z 1120.594,A -85,B 0,C 180,E1 737.953,E2 737.953} C_VEL
LIN {X 0,Y 762.232,Z 1098.376,A -85,B 0,C 180,E1 739.456,E2 739.456} C_VEL
LIN {X 0,Y 762.267,Z 1072.098,A -85,B 0,C 180,E1 740.629,E2 740.629} C_VEL
LIN {X 0,Y 762.292,Z 1043.409,A -85,B 0,C 180,E1 741.391,E2 741.391} C_VEL
LIN {X 0,Y 761.714,Z 977.53,A -85,B 0,C 180,E1 742.137,E2 742.137} C_VEL
LIN {X 0,Y 761.814,Z 977.53,A -85,B 0,C 180,E1 744.695,E2 744.695} C_VEL
LIN {X 0,Y 761.756,Z 977.53,A -85,B 0,C 180,E1 748.916,E2 748.916} C_VEL
LIN {X 0,Y 761.699,Z 977.53,A -85,B 0,C 180,E1 753.321,E2 753.321} C_VEL
LIN {X 0,Y 761.801,Z 977.53,A -85,B 0,C 180,E1 758.074,E2 758.074} C_VEL
LIN {X 0,Y 761.899,Z 977.53,A -85,B 0,C 180,E1 762.613,E2 762.613} C_VEL
LIN {X 0,Y 761.816,Z 977.53,A -85,B 0,C 180,E1 765.873,E2 765.873} C_VEL
LIN {X 0,Y 761.902,Z 977.53,A -85,B 0,C 180,E1 770.867,E2 770.867} C_VEL
LIN {X 0,Y 761.717,Z 977.53,A -85,B 0,C 180,E1 776.145,E2 776.145} C_VEL
LIN {X 0,Y 761.798,Z 977.53,A -85,B 0,C 180,E1 780.175,E2 780.175} C_VEL
LIN {X 0,Y 762.02,Z 977.53,A -85,B 0,C 180,E1 784.052,E2 784.052} C_VEL
LIN {X 0,Y 761.758,Z 977.53,A -85,B 0,C 180,E1 789.014,E2 789.014} C_VEL
LIN {X 0,Y 761.813,Z 977.53,A -85,B 0,C 180,E1 793.826,E2 793.826} C_VEL
LIN {X 0,Y 761.709,Z 977.53,A -85,B 0,C 180,E1 798.52,E2 798.52} C_VEL
LIN {X 0,Y 761.76,Z 977.53,A -85,B 0,C 180,E1 801.991,E2 801.991} C_VEL
LIN {X 0,Y 761.948,Z 977.53,A -85,B 0,C 180,E1 806.574,E2 806.574} C_VEL
LIN {X 0,Y 762.086,Z 977.53,A -85,B 0,C 180,E1 811.134,E2 811.134} C_VEL
LIN {X 0,Y 761.808,Z 977.53,A -85,B 0,C 180,E1 815.702,E2 815.702} C_VEL
LIN {X 0,Y 761.857,Z 977.53,A -85,B 0,C 180,E1 819.15,E2 819.15} C_VEL
LIN {X 0,Y 761.69,Z 977.53,A -85,B 0,C 180,E1 823.806,E2 823.806} C_VEL
LIN {X 0,Y 761.803,Z 977.53,A -85,B 0,C 180,E1 827.353,E2 827.353} C_VEL
LIN {X 0,Y 761.751,Z 977.53,A -85,B 0,C 180,E1 830.975,E2 830.975} C_VEL
LIN {X 0,Y 761.779,Z 977.53,A -85,B 0,C 180,E1 834.684,E2 834.684} C_VEL
LIN {X 0,Y 761.738,Z 977.53,A -85,B 0,C 180,E1 838.92,E2 838.92} C_VEL
LIN {X 0,Y 761.752,Z 977.53,A -85,B 0,C 180,E1 843.332,E2 843.332} C_VEL
LIN {X 0,Y 761.812,Z 977.53,A -85,B 0,C 180,E1 848.061,E2 848.061} C_VEL
LIN {X 0,Y 761.922,Z 977.53,A -85,B 0,C 180,E1 852.618,E2 852.618} C_VEL
LIN {X 0,Y 761.813,Z 977.53,A -85,B 0,C 180,E1 855.876,E2 855.876} C_VEL
LIN {X 0,Y 761.892,Z 977.53,A -85,B 0,C 180,E1 860.854,E2 860.854} C_VEL
LIN {X 0,Y 761.738,Z 977.53,A -85,B 0,C 180,E1 866.147,E2 866.147} C_VEL
LIN {X 0,Y 761.793,Z 977.53,A -85,B 0,C 180,E1 870.175,E2 870.175} C_VEL
LIN {X 0,Y 762.074,Z 977.53,A -85,B 0,C 180,E1 874.054,E2 874.054} C_VEL
LIN {X 0,Y 761.696,Z 977.53,A -85,B 0,C 180,E1 877.053,E2 877.053} C_VEL
LIN {X 0,Y 762.673,Z 1026.659,A -85,B 0,C 180,E1 877.777,E2 877.777} C_VEL
LIN {X 0,Y 762.519,Z 1065.22,A -85,B 0,C 180,E1 878.768,E2 878.768} C_VEL
LIN {X 0,Y 762.448,Z 1101.874,A -85,B 0,C 180,E1 880.172,E2 880.172} C_VEL
LIN {X 0,Y 762.325,Z 1135.773,A -85,B 0,C 180,E1 881.945,E2 881.945} C_VEL
LIN {X 0,Y 762.235,Z 1167.398,A -85,B 0,C 180,E1 884.13,E2 884.13} C_VEL
LIN {X 0,Y 762.201,Z 1195.603,A -85,B 0,C 180,E1 886.713,E2 886.713} C_VEL
LIN {X 0,Y 762.156,Z 1217.494,A -85,B 0,C 180,E1 889.396,E2 889.396} C_VEL
LIN {X 0,Y 762.092,Z 1234.425,A -85,B 0,C 180,E1 892.28,E2 892.28} C_VEL
LIN {X 0,Y 762.08,Z 1242.862,A -85,B 0,C 180,E1 894.327,E2 894.327} C_VEL
LIN {X 0,Y 759.549,Z 1245.909,A -85,B 0,C 180,E1 895.272,E2 895.272} C_VEL
LIN {X 0,Y 754.117,Z 1249.507,A -85,B 0,C 180,E1 896.779,E2 896.779} C_VEL
LIN {X 0,Y 754.098,Z 1249.552,A -85,B 0,C 180,E1 896.862,E2 896.862} C_VEL
LIN {X 0,Y 754.129,Z 1252.496,A -85,B 0,C 180,E1 899.992,E2 899.992} C_VEL
LIN {X 0,Y 754.229,Z 1250.837,A -85,B 0,C 180,E1 902.294,E2 902.294} C_VEL
LIN {X 0,Y 754.239,Z 1244.399,A -85,B 0,C 180,E1 905.178,E2 905.178} C_VEL
LIN {X 0,Y 754.185,Z 1232.678,A -85,B 0,C 180,E1 908.076,E2 908.076} C_VEL
LIN {X 0,Y 754.302,Z 1214.918,A -85,B 0,C 180,E1 910.992,E2 910.992} C_VEL
LIN {X 0,Y 754.401,Z 1191.613,A -85,B 0,C 180,E1 913.751,E2 913.751} C_VEL
LIN {X 0,Y 754.525,Z 1164.238,A -85,B 0,C 180,E1 916.193,E2 916.193} C_VEL
LIN {X 0,Y 754.731,Z 1132.56,A -85,B 0,C 180,E1 918.347,E2 918.347} C_VEL
LIN {X 0,Y 754.908,Z 1096.073,A -85,B 0,C 180,E1 920.207,E2 920.207} C_VEL
LIN {X 0,Y 755.146,Z 1056.744,A -85,B 0,C 180,E1 921.625,E2 921.625} C_VEL
LIN {X 0,Y 755.216,Z 1017.586,A -85,B 0,C 180,E1 922.538,E2 922.538} C_VEL
LIN {X 0,Y 754.479,Z 979.861,A -85,B 0,C 180,E1 923.037,E2 923.037} C_VEL
LIN {X 0,Y 754.198,Z 977.53,A -85,B 0,C 180,E1 923.105,E2 923.105} C_VEL
LIN {X 0,Y 753.87,Z 977.53,A -85,B 0,C 180,E1 928.829,E2 928.829} C_VEL
LIN {X 0,Y 753.948,Z 977.53,A -85,B 0,C 180,E1 932.849,E2 932.849} C_VEL
LIN {X 0,Y 754.123,Z 977.53,A -85,B 0,C 180,E1 937.055,E2 937.055} C_VEL
LIN {X 0,Y 753.763,Z 977.53,A -85,B 0,C 180,E1 943.099,E2 943.099} C_VEL
LIN {X 0,Y 753.675,Z 977.53,A -85,B 0,C 180,E1 948.443,E2 948.443} C_VEL
LIN {X 0,Y 754.008,Z 977.53,A -85,B 0,C 180,E1 953.476,E2 953.476} C_VEL
LIN {X 0,Y 753.681,Z 977.53,A -85,B 0,C 180,E1 958.491,E2 958.491} C_VEL
LIN {X 0,Y 753.762,Z 977.53,A -85,B 0,C 180,E1 962.466,E2 962.466} C_VEL
LIN {X 0,Y 754.136,Z 977.53,A -85,B 0,C 180,E1 966.263,E2 966.263} C_VEL
LIN {X 0,Y 755.251,Z 1027.959,A -85,B 0,C 180,E1 966.822,E2 966.822} C_VEL
LIN {X 0,Y 755.267,Z 1080.64,A -85,B 0,C 180,E1 967.474,E2 967.474} C_VEL
LIN {X 0,Y 755.148,Z 1120.573,A -85,B 0,C 180,E1 968.447,E2 968.447} C_VEL
LIN {X 0,Y 754.931,Z 1158.42,A -85,B 0,C 180,E1 969.854,E2 969.854} C_VEL
LIN {X 0,Y 754.702,Z 1193.229,A -85,B 0,C 180,E1 971.647,E2 971.647} C_VEL
LIN {X 0,Y 754.516,Z 1224.689,A -85,B 0,C 180,E1 973.797,E2 973.797} C_VEL
LIN {X 0,Y 754.374,Z 1251.842,A -85,B 0,C 180,E1 976.226,E2 976.226} C_VEL
LIN {X 0,Y 754.29,Z 1275.217,A -85,B 0,C 180,E1 979.004,E2 979.004} C_VEL
LIN {X 0,Y 754.214,Z 1292.899,A -85,B 0,C 180,E1 981.921,E2 981.921} C_VEL
LIN {X 0,Y 754.225,Z 1304.534,A -85,B 0,C 180,E1 984.818,E2 984.818} C_VEL
LIN {X 0,Y 754.159,Z 1310.902,A -85,B 0,C 180,E1 987.702,E2 987.702} C_VEL
LIN {X 0,Y 754.101,Z 1312.5,A -85,B 0,C 180,E1 990.005,E2 990.005} C_VEL
LIN {X 0,Y 754.174,Z 1310.886,A -85,B 0,C 180,E1 992.308,E2 992.308} C_VEL
LIN {X 0,Y 754.225,Z 1304.499,A -85,B 0,C 180,E1 995.192,E2 995.192} C_VEL
LIN {X 0,Y 754.206,Z 1292.842,A -85,B 0,C 180,E1 998.09,E2 998.09} C_VEL
LIN {X 0,Y 754.282,Z 1275.136,A -85,B 0,C 180,E1 1001.007,E2 1001.007} C_VEL
LIN {X 0,Y 754.383,Z 1251.796,A -85,B 0,C 180,E1 1003.779,E2 1003.779} C_VEL
LIN {X 0,Y 754.527,Z 1224.731,A -85,B 0,C 180,E1 1006.199,E2 1006.199} C_VEL
LIN {X 0,Y 754.709,Z 1193.043,A -85,B 0,C 180,E1 1008.364,E2 1008.364} C_VEL
LIN {X 0,Y 754.915,Z 1158.192,A -85,B 0,C 180,E1 1010.157,E2 1010.157} C_VEL
LIN {X 0,Y 755.156,Z 1120.213,A -85,B 0,C 180,E1 1011.564,E2 1011.564} C_VEL
LIN {X 0,Y 755.299,Z 1080.294,A -85,B 0,C 180,E1 1012.532,E2 1012.532} C_VEL
LIN {X 0,Y 755.181,Z 1026.994,A -85,B 0,C 180,E1 1013.19,E2 1013.19} C_VEL
LIN {X 0,Y 754.1,Z 977.53,A -85,B 0,C 180,E1 1013.754,E2 1013.754} C_VEL
LIN {X 0,Y 753.874,Z 977.53,A -85,B 0,C 180,E1 1018.848,E2 1018.848} C_VEL
LIN {X 0,Y 753.915,Z 977.53,A -85,B 0,C 180,E1 1022.871,E2 1022.871} C_VEL
LIN {X 0,Y 754.137,Z 977.53,A -85,B 0,C 180,E1 1027.076,E2 1027.076} C_VEL
LIN {X 0,Y 753.984,Z 977.53,A -85,B 0,C 180,E1 1033.108,E2 1033.108} C_VEL
LIN {X 0,Y 753.603,Z 977.53,A -85,B 0,C 180,E1 1036.889,E2 1036.889} C_VEL
LIN {X 0,Y 753.742,Z 977.53,A -85,B 0,C 180,E1 1041.639,E2 1041.639} C_VEL
LIN {X 0,Y 753.768,Z 977.53,A -85,B 0,C 180,E1 1045.76,E2 1045.76} C_VEL
LIN {X 0,Y 753.892,Z 977.53,A -85,B 0,C 180,E1 1049.849,E2 1049.849} C_VEL
LIN {X 0,Y 753.908,Z 977.53,A -85,B 0,C 180,E1 1054.761,E2 1054.761} C_VEL
LIN {X 0,Y 753.897,Z 977.53,A -85,B 0,C 180,E1 1058.802,E2 1058.802} C_VEL
LIN {X 0,Y 753.906,Z 977.53,A -85,B 0,C 180,E1 1063.668,E2 1063.668} C_VEL
LIN {X 0,Y 753.765,Z 977.53,A -85,B 0,C 180,E1 1068.413,E2 1068.413} C_VEL
LIN {X 0,Y 754.086,Z 977.53,A -85,B 0,C 180,E1 1073.084,E2 1073.084} C_VEL
LIN {X 0,Y 754.141,Z 977.53,A -85,B 0,C 180,E1 1077.669,E2 1077.669} C_VEL
LIN {X 0,Y 754.61,Z 1042.831,A -85,B 0,C 180,E1 1078.39,E2 1078.39} C_VEL
LIN {X 0,Y 754.536,Z 1071.369,A -85,B 0,C 180,E1 1079.145,E2 1079.145} C_VEL
LIN {X 0,Y 754.48,Z 1097.26,A -85,B 0,C 180,E1 1080.296,E2 1080.296} C_VEL
LIN {X 0,Y 754.394,Z 1118.857,A -85,B 0,C 180,E1 1081.735,E2 1081.735} C_VEL
LIN {X 0,Y 754.343,Z 1137.001,A -85,B 0,C 180,E1 1083.463,E2 1083.463} C_VEL
LIN {X 0,Y 754.32,Z 1150.916,A -85,B 0,C 180,E1 1085.483,E2 1085.483} C_VEL
LIN {X 0,Y 754.306,Z 1159.106,A -85,B 0,C 180,E1 1087.51,E2 1087.51} C_VEL
LIN {X 0,Y 754.245,Z 1162.199,A -85,B 0,C 180,E1 1089.256,E2 1089.256} C_VEL
LIN {X 0,Y 754.272,Z 1162.371,A -85,B 0,C 180,E1 1090.424,E2 1090.424} C_VEL
LIN {X 0,Y 754.291,Z 1159.686,A -85,B 0,C 180,E1 1092.184,E2 1092.184} C_VEL
LIN {X 0,Y 754.32,Z 1151.844,A -85,B 0,C 180,E1 1094.252,E2 1094.252} C_VEL
LIN {X 0,Y 754.316,Z 1137.897,A -85,B 0,C 180,E1 1096.34,E2 1096.34} C_VEL
LIN {X 0,Y 754.342,Z 1119.221,A -85,B 0,C 180,E1 1098.147,E2 1098.147} C_VEL
LIN {X 0,Y 754.411,Z 1098.092,A -85,B 0,C 180,E1 1099.571,E2 1099.571} C_VEL
LIN {X 0,Y 754.514,Z 1071.779,A -85,B 0,C 180,E1 1100.751,E2 1100.751} C_VEL
LIN {X 0,Y 754.562,Z 1043.935,A -85,B 0,C 180,E1 1101.5,E2 1101.5} C_VEL
LIN {X 0,Y 754.039,Z 977.53,A -85,B 0,C 180,E1 1102.278,E2 1102.278} C_VEL
LIN {X 0,Y 753.759,Z 977.53,A -85,B 0,C 180,E1 1106.254,E2 1106.254} C_VEL
LIN {X 0,Y 753.709,Z 977.53,A -85,B 0,C 180,E1 1110.178,E2 1110.178} C_VEL
LIN {X 0,Y 753.948,Z 977.53,A -85,B 0,C 180,E1 1112.869,E2 1112.869} C_VEL
LIN {X 0,Y 754.128,Z 977.53,A -85,B 0,C 180,E1 1117.075,E2 1117.075} C_VEL
LIN {X 0,Y 753.972,Z 977.53,A -85,B 0,C 180,E1 1123.107,E2 1123.107} C_VEL
LIN {X 0,Y 753.619,Z 977.53,A -85,B 0,C 180,E1 1126.866,E2 1126.866} C_VEL
LIN {X 0,Y 753.742,Z 977.53,A -85,B 0,C 180,E1 1131.635,E2 1131.635} C_VEL
LIN {X 0,Y 753.779,Z 977.53,A -85,B 0,C 180,E1 1135.74,E2 1135.74} C_VEL
LIN {X 0,Y 753.918,Z 977.53,A -85,B 0,C 180,E1 1139.831,E2 1139.831} C_VEL
LIN {X 0,Y 753.901,Z 977.53,A -85,B 0,C 180,E1 1144.755,E2 1144.755} C_VEL
LIN {X 0,Y 753.895,Z 977.53,A -85,B 0,C 180,E1 1148.784,E2 1148.784} C_VEL
LIN {X 0,Y 753.909,Z 977.53,A -85,B 0,C 180,E1 1153.652,E2 1153.652} C_VEL
LIN {X 0,Y 753.788,Z 977.53,A -85,B 0,C 180,E1 1158.398,E2 1158.398} C_VEL
LIN {X 0,Y 753.854,Z 977.53,A -85,B 0,C 180,E1 1161.906,E2 1161.906} C_VEL
LIN {X 0,Y 754.047,Z 977.53,A -85,B 0,C 180,E1 1166.538,E2 1166.538} C_VEL
LIN {X 0,Y 754.18,Z 977.53,A -85,B 0,C 180,E1 1171.146,E2 1171.146} C_VEL
LIN {X 0,Y 753.919,Z 977.53,A -85,B 0,C 180,E1 1175.762,E2 1175.762} C_VEL
LIN {X 0,Y 753.823,Z 977.53,A -85,B 0,C 180,E1 1180.417,E2 1180.417} C_VEL
LIN {X 0,Y 753.783,Z 977.53,A -85,B 0,C 180,E1 1183.953,E2 1183.953} C_VEL
LIN {X 0,Y 753.873,Z 977.53,A -85,B 0,C 180,E1 1187.542,E2 1187.542} C_VEL
LIN {X 0,Y 753.816,Z 977.53,A -85,B 0,C 180,E1 1191.206,E2 1191.206} C_VEL
LIN {X 0,Y 753.784,Z 977.53,A -85,B 0,C 180,E1 1195.226,E2 1195.226} C_VEL
LIN {X 0,Y 753.856,Z 977.53,A -85,B 0,C 180,E1 1198.836,E2 1198.836} C_VEL
LIN {X 0,Y 753.976,Z 977.53,A -85,B 0,C 180,E1 1202.856,E2 1202.856} C_VEL
LIN {X 0,Y 754.141,Z 977.53,A -85,B 0,C 180,E1 1207.062,E2 1207.062} C_VEL
LIN {X 0,Y 753.983,Z 977.53,A -85,B 0,C 180,E1 1213.094,E2 1213.094} C_VEL
LIN {X 0,Y 753.638,Z 977.53,A -85,B 0,C 180,E1 1216.869,E2 1216.869} C_VEL
LIN {X 0,Y 753.771,Z 977.53,A -85,B 0,C 180,E1 1221.619,E2 1221.619} C_VEL
LIN {X 0,Y 753.791,Z 977.53,A -85,B 0,C 180,E1 1225.741,E2 1225.741} C_VEL
LIN {X 0,Y 753.903,Z 977.53,A -85,B 0,C 180,E1 1229.831,E2 1229.831} C_VEL
LIN {X 0,Y 753.945,Z 977.53,A -85,B 0,C 180,E1 1235.03,E2 1235.03} C_VEL
LIN {X 0,Y 754.136,Z 977.53,A -85,B 0,C 180,E1 1236.821,E2 1236.821} C_VEL
LIN {X 0,Y 755.34,Z 1025.167,A -85,B 0,C 180,E1 1237.521,E2 1237.521} C_VEL
LIN {X 0,Y 755.101,Z 1064.003,A -85,B 0,C 180,E1 1238.511,E2 1238.511} C_VEL
LIN {X 0,Y 754.909,Z 1100.655,A -85,B 0,C 180,E1 1239.911,E2 1239.911} C_VEL
LIN {X 0,Y 754.699,Z 1135.013,A -85,B 0,C 180,E1 1241.71,E2 1241.71} C_VEL
LIN {X 0,Y 754.496,Z 1165.351,A -85,B 0,C 180,E1 1243.804,E2 1243.804} C_VEL
LIN {X 0,Y 754.382,Z 1192.347,A -85,B 0,C 180,E1 1246.232,E2 1246.232} C_VEL
LIN {X 0,Y 754.329,Z 1215.463,A -85,B 0,C 180,E1 1248.992,E2 1248.992} C_VEL
LIN {X 0,Y 754.251,Z 1233.097,A -85,B 0,C 180,E1 1251.916,E2 1251.916} C_VEL
LIN {X 0,Y 754.251,Z 1244.642,A -85,B 0,C 180,E1 1254.806,E2 1254.806} C_VEL
LIN {X 0,Y 754.098,Z 1249.552,A -85,B 0,C 180,E1 1256.862,E2 1256.862} C_VEL
LIN {X 0,Y 752.869,Z 1250.694,A -85,B 0,C 180,E1 1257.514,E2 1257.514} C_VEL
LIN {X 0,Y 746.276,Z 1252.316,A -85,B 0,C 180,E1 1259.289,E2 1259.289} C_VEL
LIN {X 0,Y 746.187,Z 1252.32,A -85,B 0,C 180,E1 1259.457,E2 1259.457} C_VEL
LIN {X 0,Y 746.326,Z 1250.838,A -85,B 0,C 180,E1 1262.319,E2 1262.319} C_VEL
LIN {X 0,Y 746.361,Z 1244.401,A -85,B 0,C 180,E1 1265.233,E2 1265.233} C_VEL
LIN {X 0,Y 746.303,Z 1232.68,A -85,B 0,C 180,E1 1268.161,E2 1268.161} C_VEL
LIN {X 0,Y 746.434,Z 1214.924,A -85,B 0,C 180,E1 1271.109,E2 1271.109} C_VEL
LIN {X 0,Y 746.588,Z 1192.659,A -85,B 0,C 180,E1 1273.792,E2 1273.792} C_VEL
LIN {X 0,Y 746.811,Z 1165.488,A -85,B 0,C 180,E1 1276.266,E2 1276.266} C_VEL
LIN {X 0,Y 747.093,Z 1135.072,A -85,B 0,C 180,E1 1278.388,E2 1278.388} C_VEL
LIN {X 0,Y 747.352,Z 1100.51,A -85,B 0,C 180,E1 1280.218,E2 1280.218} C_VEL
LIN {X 0,Y 747.672,Z 1062.972,A -85,B 0,C 180,E1 1281.656,E2 1281.656} C_VEL
LIN {X 0,Y 747.904,Z 1023.672,A -85,B 0,C 180,E1 1282.655,E2 1282.655} C_VEL
LIN {X 0,Y 747.253,Z 981.417,A -85,B 0,C 180,E1 1283.258,E2 1283.258} C_VEL
LIN {X 0,Y 746.207,Z 977.53,A -85,B 0,C 180,E1 1283.384,E2 1283.384} C_VEL
LIN {X 0,Y 745.89,Z 977.53,A -85,B 0,C 180,E1 1289.167,E2 1289.167} C_VEL
LIN {X 0,Y 745.857,Z 977.53,A -85,B 0,C 180,E1 1293.608,E2 1293.608} C_VEL
LIN {X 0,Y 746.031,Z 977.53,A -85,B 0,C 180,E1 1297.624,E2 1297.624} C_VEL
LIN {X 0,Y 745.852,Z 977.53,A -85,B 0,C 180,E1 1303.007,E2 1303.007} C_VEL
LIN {X 0,Y 745.851,Z 977.53,A -85,B 0,C 180,E1 1307.908,E2 1307.908} C_VEL
LIN {X 0,Y 746.093,Z 977.53,A -85,B 0,C 180,E1 1312.469,E2 1312.469} C_VEL
LIN {X 0,Y 745.912,Z 977.53,A -85,B 0,C 180,E1 1316.743,E2 1316.743} C_VEL
LIN {X 0,Y 745.928,Z 977.53,A -85,B 0,C 180,E1 1322.152,E2 1322.152} C_VEL
LIN {X 0,Y 746.148,Z 977.968,A -85,B 0,C 180,E1 1326.007,E2 1326.007} C_VEL
LIN {X 0,Y 747.794,Z 989.059,A -85,B 0,C 180,E1 1326.178,E2 1326.178} C_VEL
LIN {X 0,Y 747.987,Z 1076.593,A -85,B 0,C 180,E1 1327.169,E2 1327.169} C_VEL
LIN {X 0,Y 747.788,Z 1116.8,A -85,B 0,C 180,E1 1328.107,E2 1328.107} C_VEL
LIN {X 0,Y 747.467,Z 1155.579,A -85,B 0,C 180,E1 1329.515,E2 1329.515} C_VEL
LIN {X 0,Y 747.128,Z 1191.983,A -85,B 0,C 180,E1 1331.377,E2 1331.377} C_VEL
LIN {X 0,Y 746.808,Z 1223.141,A -85,B 0,C 180,E1 1333.503,E2 1333.503} C_VEL
LIN {X 0,Y 746.547,Z 1250.183,A -85,B 0,C 180,E1 1335.909,E2 1335.909} C_VEL
LIN {X 0,Y 746.4,Z 1273.027,A -85,B 0,C 180,E1 1338.589,E2 1338.589} C_VEL
LIN {X 0,Y 746.274,Z 1289.827,A -85,B 0,C 180,E1 1341.246,E2 1341.246} C_VEL
LIN {X 0,Y 746.256,Z 1302.616,A -85,B 0,C 180,E1 1344.178,E2 1344.178} C_VEL
LIN {X 0,Y 746.226,Z 1308.943,A -85,B 0,C 180,E1 1346.513,E2 1346.513} C_VEL
LIN {X 0,Y 746.265,Z 1312.09,A -85,B 0,C 180,E1 1348.842,E2 1348.842} C_VEL
LIN {X 0,Y 746.237,Z 1312.081,A -85,B 0,C 180,E1 1351.169,E2 1351.169} C_VEL
LIN {X 0,Y 746.28,Z 1307.696,A -85,B 0,C 180,E1 1354.081,E2 1354.081} C_VEL
LIN {X 0,Y 746.35,Z 1296.91,A -85,B 0,C 180,E1 1357.295,E2 1357.295} C_VEL
LIN {X 0,Y 746.384,Z 1280.491,A -85,B 0,C 180,E1 1360.333,E2 1360.333} C_VEL
LIN {X 0,Y 746.524,Z 1259.527,A -85,B 0,C 180,E1 1363.088,E2 1363.088} C_VEL
LIN {X 0,Y 746.751,Z 1233.617,A -85,B 0,C 180,E1 1365.637,E2 1365.637} C_VEL
LIN {X 0,Y 746.974,Z 1203.952,A -85,B 0,C 180,E1 1367.873,E2 1367.873} C_VEL
LIN {X 0,Y 747.28,Z 1170.025,A -85,B 0,C 180,E1 1369.814,E2 1369.814} C_VEL
LIN {X 0,Y 747.618,Z 1132.079,A -85,B 0,C 180,E1 1371.402,E2 1371.402} C_VEL
LIN {X 0,Y 747.921,Z 1092.161,A -85,B 0,C 180,E1 1372.528,E2 1372.528} C_VEL
LIN {X 0,Y 748.025,Z 1050.563,A -85,B 0,C 180,E1 1373.184,E2 1373.184} C_VEL
LIN {X 0,Y 746.813,Z 980.727,A -85,B 0,C 180,E1 1373.941,E2 1373.941} C_VEL
LIN {X 0,Y 746.096,Z 977.53,A -85,B 0,C 180,E1 1374.043,E2 1374.043} C_VEL
LIN {X 0,Y 745.895,Z 977.53,A -85,B 0,C 180,E1 1379.186,E2 1379.186} C_VEL
LIN {X 0,Y 745.841,Z 977.53,A -85,B 0,C 180,E1 1383.621,E2 1383.621} C_VEL
LIN {X 0,Y 746.043,Z 977.53,A -85,B 0,C 180,E1 1387.639,E2 1387.639} C_VEL
LIN {X 0,Y 746.123,Z 977.53,A -85,B 0,C 180,E1 1393.676,E2 1393.676} C_VEL
LIN {X 0,Y 745.83,Z 977.53,A -85,B 0,C 180,E1 1399.466,E2 1399.466} C_VEL
LIN {X 0,Y 745.854,Z 977.53,A -85,B 0,C 180,E1 1404.363,E2 1404.363} C_VEL
LIN {X 0,Y 745.975,Z 977.53,A -85,B 0,C 180,E1 1409.495,E2 1409.495} C_VEL
LIN {X 0,Y 746.031,Z 977.53,A -85,B 0,C 180,E1 1414.765,E2 1414.765} C_VEL
LIN {X 0,Y 745.927,Z 977.53,A -85,B 0,C 180,E1 1419.152,E2 1419.152} C_VEL
LIN {X 0,Y 746.001,Z 977.53,A -85,B 0,C 180,E1 1423.49,E2 1423.49} C_VEL
LIN {X 0,Y 745.844,Z 977.53,A -85,B 0,C 180,E1 1428.288,E2 1428.288} C_VEL
LIN {X 0,Y 746.178,Z 977.53,A -85,B 0,C 180,E1 1433.011,E2 1433.011} C_VEL
LIN {X 0,Y 746.219,Z 977.53,A -85,B 0,C 180,E1 1437.536,E2 1437.536} C_VEL
LIN {X 0,Y 746.891,Z 1042.59,A -85,B 0,C 180,E1 1438.265,E2 1438.265} C_VEL
LIN {X 0,Y 746.767,Z 1071.238,A -85,B 0,C 180,E1 1439.027,E2 1439.027} C_VEL
LIN {X 0,Y 746.655,Z 1097.847,A -85,B 0,C 180,E1 1440.226,E2 1440.226} C_VEL
LIN {X 0,Y 746.538,Z 1120.185,A -85,B 0,C 180,E1 1441.753,E2 1441.753} C_VEL
LIN {X 0,Y 746.446,Z 1139.08,A -85,B 0,C 180,E1 1443.645,E2 1443.645} C_VEL
LIN {X 0,Y 746.417,Z 1151.972,A -85,B 0,C 180,E1 1445.636,E2 1445.636} C_VEL
LIN {X 0,Y 746.405,Z 1159.388,A -85,B 0,C 180,E1 1447.59,E2 1447.59} C_VEL
LIN {X 0,Y 746.342,Z 1162.291,A -85,B 0,C 180,E1 1449.355,E2 1449.355} C_VEL
LIN {X 0,Y 746.353,Z 1160.76,A -85,B 0,C 180,E1 1451.721,E2 1451.721} C_VEL
LIN {X 0,Y 746.373,Z 1154.294,A -85,B 0,C 180,E1 1453.778,E2 1453.778} C_VEL
LIN {X 0,Y 746.436,Z 1141.773,A -85,B 0,C 180,E1 1455.912,E2 1455.912} C_VEL
LIN {X 0,Y 746.5,Z 1125.139,A -85,B 0,C 180,E1 1457.733,E2 1457.733} C_VEL
LIN {X 0,Y 746.627,Z 1103.08,A -85,B 0,C 180,E1 1459.379,E2 1459.379} C_VEL
LIN {X 0,Y 746.736,Z 1077.348,A -85,B 0,C 180,E1 1460.656,E2 1460.656} C_VEL
LIN {X 0,Y 746.836,Z 1048.141,A -85,B 0,C 180,E1 1461.536,E2 1461.536} C_VEL
LIN {X 0,Y 746.805,Z 1012.238,A -85,B 0,C 180,E1 1462.014,E2 1462.014} C_VEL
LIN {X 0,Y 746.213,Z 977.53,A -85,B 0,C 180,E1 1462.401,E2 1462.401} C_VEL
LIN {X 0,Y 745.977,Z 977.53,A -85,B 0,C 180,E1 1467.858,E2 1467.858} C_VEL
LIN {X 0,Y 745.916,Z 977.53,A -85,B 0,C 180,E1 1473.268,E2 1473.268} C_VEL
LIN {X 0,Y 746.048,Z 977.53,A -85,B 0,C 180,E1 1477.608,E2 1477.608} C_VEL
LIN {X 0,Y 746.088,Z 977.53,A -85,B 0,C 180,E1 1483.676,E2 1483.676} C_VEL
LIN {X 0,Y 745.717,Z 977.53,A -85,B 0,C 180,E1 1488.753,E2 1488.753} C_VEL
LIN {X 0,Y 745.738,Z 977.53,A -85,B 0,C 180,E1 1492.435,E2 1492.435} C_VEL
LIN {X 0,Y 745.781,Z 977.53,A -85,B 0,C 180,E1 1496.724,E2 1496.724} C_VEL
LIN {X 0,Y 745.839,Z 977.53,A -85,B 0,C 180,E1 1500.884,E2 1500.884} C_VEL
LIN {X 0,Y 746.028,Z 977.53,A -85,B 0,C 180,E1 1504.746,E2 1504.746} C_VEL
LIN {X 0,Y 745.931,Z 977.53,A -85,B 0,C 180,E1 1509.142,E2 1509.142} C_VEL
LIN {X 0,Y 746.001,Z 977.53,A -85,B 0,C 180,E1 1513.473,E2 1513.473} C_VEL
LIN {X 0,Y 745.868,Z 977.53,A -85,B 0,C 180,E1 1518.273,E2 1518.273} C_VEL
LIN {X 0,Y 746.187,Z 977.53,A -85,B 0,C 180,E1 1522.996,E2 1522.996} C_VEL
LIN {X 0,Y 746.169,Z 977.53,A -85,B 0,C 180,E1 1527.667,E2 1527.667} C_VEL
LIN {X 0,Y 746.003,Z 977.53,A -85,B 0,C 180,E1 1532.323,E2 1532.323} C_VEL
LIN {X 0,Y 746.011,Z 977.53,A -85,B 0,C 180,E1 1535.823,E2 1535.823} C_VEL
LIN {X 0,Y 745.922,Z 977.53,A -85,B 0,C 180,E1 1540.529,E2 1540.529} C_VEL
LIN {X 0,Y 746.03,Z 977.53,A -85,B 0,C 180,E1 1545.304,E2 1545.304} C_VEL
LIN {X 0,Y 746.086,Z 977.53,A -85,B 0,C 180,E1 1550.192,E2 1550.192} C_VEL
LIN {X 0,Y 745.906,Z 977.53,A -85,B 0,C 180,E1 1555.246,E2 1555.246} C_VEL
LIN {X 0,Y 745.898,Z 977.53,A -85,B 0,C 180,E1 1559.173,E2 1559.173} C_VEL
LIN {X 0,Y 745.895,Z 977.53,A -85,B 0,C 180,E1 1563.597,E2 1563.597} C_VEL
LIN {X 0,Y 746.048,Z 977.53,A -85,B 0,C 180,E1 1567.612,E2 1567.612} C_VEL
LIN {X 0,Y 746.088,Z 977.53,A -85,B 0,C 180,E1 1573.664,E2 1573.664} C_VEL
LIN {X 0,Y 745.723,Z 977.53,A -85,B 0,C 180,E1 1578.74,E2 1578.74} C_VEL
LIN {X 0,Y 745.767,Z 977.53,A -85,B 0,C 180,E1 1582.438,E2 1582.438} C_VEL
LIN {X 0,Y 745.78,Z 977.53,A -85,B 0,C 180,E1 1586.725,E2 1586.725} C_VEL
LIN {X 0,Y 745.833,Z 977.53,A -85,B 0,C 180,E1 1590.869,E2 1590.869} C_VEL
LIN {X 0,Y 746.131,Z 977.53,A -85,B 0,C 180,E1 1594.75,E2 1594.75} C_VEL
LIN {X 0,Y 746.156,Z 977.53,A -85,B 0,C 180,E1 1596.558,E2 1596.558} C_VEL
LIN {X 0,Y 747.983,Z 999.321,A -85,B 0,C 180,E1 1596.872,E2 1596.872} C_VEL
LIN {X 0,Y 747.954,Z 1038.973,A -85,B 0,C 180,E1 1597.591,E2 1597.591} C_VEL
LIN {X 0,Y 747.578,Z 1077.108,A -85,B 0,C 180,E1 1598.737,E2 1598.737} C_VEL
LIN {X 0,Y 747.275,Z 1112.687,A -85,B 0,C 180,E1 1600.277,E2 1600.277} C_VEL
LIN {X 0,Y 746.978,Z 1145.736,A -85,B 0,C 180,E1 1602.202,E2 1602.202} C_VEL
LIN {X 0,Y 746.706,Z 1174.614,A -85,B 0,C 180,E1 1604.402,E2 1604.402} C_VEL
LIN {X 0,Y 746.498,Z 1200.377,A -85,B 0,C 180,E1 1606.962,E2 1606.962} C_VEL
LIN {X 0,Y 746.368,Z 1222.121,A -85,B 0,C 180,E1 1609.868,E2 1609.868} C_VEL
LIN {X 0,Y 746.29,Z 1237.1,A -85,B 0,C 180,E1 1612.702,E2 1612.702} C_VEL
LIN {X 0,Y 746.233,Z 1247.804,A -85,B 0,C 180,E1 1615.917,E2 1615.917} C_VEL
LIN {X 0,Y 746.22,Z 1252.113,A -85,B 0,C 180,E1 1618.828,E2 1618.828} C_VEL
LIN {X 0,Y 746.187,Z 1252.32,A -85,B 0,C 180,E1 1619.457,E2 1619.457} C_VEL
LIN {X 0,Y 744.957,Z 1252.459,A -85,B 0,C 180,E1 1620.124,E2 1620.124} C_VEL
LIN {X 0,Y 738.435,Z 1251.306,A -85,B 0,C 180,E1 1622.017,E2 1622.017} C_VEL
LIN {X 0,Y 738.418,Z 1251.087,A -85,B 0,C 180,E1 1622.102,E2 1622.102} C_VEL
LIN {X 0,Y 738.482,Z 1244.549,A -85,B 0,C 180,E1 1625.244,E2 1625.244} C_VEL
LIN {X 0,Y 738.424,Z 1232.681,A -85,B 0,C 180,E1 1628.249,E2 1628.249} C_VEL
LIN {X 0,Y 738.577,Z 1214.928,A -85,B 0,C 180,E1 1631.229,E2 1631.229} C_VEL
LIN {X 0,Y 738.78,Z 1192.723,A -85,B 0,C 180,E1 1633.935,E2 1633.935} C_VEL
LIN {X 0,Y 739.085,Z 1166.479,A -85,B 0,C 180,E1 1636.363,E2 1636.363} C_VEL
LIN {X 0,Y 739.488,Z 1135.081,A -85,B 0,C 180,E1 1638.584,E2 1638.584} C_VEL
LIN {X 0,Y 739.835,Z 1100.742,A -85,B 0,C 180,E1 1640.422,E2 1640.422} C_VEL
LIN {X 0,Y 740.28,Z 1064.201,A -85,B 0,C 180,E1 1641.844,E2 1641.844} C_VEL
LIN {X 0,Y 740.596,Z 1025.039,A -85,B 0,C 180,E1 1642.864,E2 1642.864} C_VEL
LIN {X 0,Y 739.929,Z 983.378,A -85,B 0,C 180,E1 1643.482,E2 1643.482} C_VEL
LIN {X 0,Y 738.196,Z 977.53,A -85,B 0,C 180,E1 1643.649,E2 1643.649} C_VEL
LIN {X 0,Y 737.931,Z 977.53,A -85,B 0,C 180,E1 1649.512,E2 1649.512} C_VEL
LIN {X 0,Y 737.948,Z 977.53,A -85,B 0,C 180,E1 1653.655,E2 1653.655} C_VEL
LIN {X 0,Y 738.004,Z 977.53,A -85,B 0,C 180,E1 1658.006,E2 1658.006} C_VEL
LIN {X 0,Y 737.95,Z 977.53,A -85,B 0,C 180,E1 1662.639,E2 1662.639} C_VEL
LIN {X 0,Y 737.948,Z 977.53,A -85,B 0,C 180,E1 1667.644,E2 1667.644} C_VEL
LIN {X 0,Y 738.091,Z 977.53,A -85,B 0,C 180,E1 1673.469,E2 1673.469} C_VEL
LIN {X 0,Y 737.923,Z 977.53,A -85,B 0,C 180,E1 1677.738,E2 1677.738} C_VEL
LIN {X 0,Y 738.019,Z 977.53,A -85,B 0,C 180,E1 1681.958,E2 1681.958} C_VEL
LIN {X 0,Y 738.095,Z 977.53,A -85,B 0,C 180,E1 1685.719,E2 1685.719} C_VEL
LIN {X 0,Y 740.517,Z 987.945,A -85,B 0,C 180,E1 1685.917,E2 1685.917} C_VEL
LIN {X 0,Y 740.666,Z 1075.371,A -85,B 0,C 180,E1 1686.91,E2 1686.91} C_VEL
LIN {X 0,Y 740.432,Z 1115.438,A -85,B 0,C 180,E1 1687.838,E2 1687.838} C_VEL
LIN {X 0,Y 740,Z 1154.127,A -85,B 0,C 180,E1 1689.235,E2 1689.235} C_VEL
LIN {X 0,Y 739.521,Z 1190.719,A -85,B 0,C 180,E1 1691.101,E2 1691.101} C_VEL
LIN {X 0,Y 739.1,Z 1223.142,A -85,B 0,C 180,E1 1693.326,E2 1693.326} C_VEL
LIN {X 0,Y 738.757,Z 1250.188,A -85,B 0,C 180,E1 1695.757,E2 1695.757} C_VEL
LIN {X 0,Y 738.555,Z 1273.025,A -85,B 0,C 180,E1 1698.466,E2 1698.466} C_VEL
LIN {X 0,Y 738.387,Z 1289.831,A -85,B 0,C 180,E1 1701.152,E2 1701.152} C_VEL
LIN {X 0,Y 738.376,Z 1302.614,A -85,B 0,C 180,E1 1704.116,E2 1704.116} C_VEL
LIN {X 0,Y 738.356,Z 1308.946,A -85,B 0,C 180,E1 1706.476,E2 1706.476} C_VEL
LIN {X 0,Y 738.364,Z 1312.093,A -85,B 0,C 180,E1 1708.83,E2 1708.83} C_VEL
LIN {X 0,Y 738.336,Z 1312.083,A -85,B 0,C 180,E1 1711.181,E2 1711.181} C_VEL
LIN {X 0,Y 738.378,Z 1307.692,A -85,B 0,C 180,E1 1714.124,E2 1714.124} C_VEL
LIN {X 0,Y 738.479,Z 1296.913,A -85,B 0,C 180,E1 1717.374,E2 1717.374} C_VEL
LIN {X 0,Y 738.526,Z 1280.419,A -85,B 0,C 180,E1 1720.456,E2 1720.456} C_VEL
LIN {X 0,Y 738.717,Z 1259.531,A -85,B 0,C 180,E1 1723.229,E2 1723.229} C_VEL
LIN {X 0,Y 739.001,Z 1234.696,A -85,B 0,C 180,E1 1725.712,E2 1725.712} C_VEL
LIN {X 0,Y 739.323,Z 1203.958,A -85,B 0,C 180,E1 1728.064,E2 1728.064} C_VEL
LIN {X 0,Y 739.759,Z 1169.827,A -85,B 0,C 180,E1 1730.035,E2 1730.035} C_VEL
LIN {X 0,Y 740.209,Z 1132.087,A -85,B 0,C 180,E1 1731.627,E2 1731.627} C_VEL
LIN {X 0,Y 740.598,Z 1092.157,A -85,B 0,C 180,E1 1732.763,E2 1732.763} C_VEL
LIN {X 0,Y 740.796,Z 1053.388,A -85,B 0,C 180,E1 1733.393,E2 1733.393} C_VEL
LIN {X 0,Y 739.748,Z 983.09,A -85,B 0,C 180,E1 1734.16,E2 1734.16} C_VEL
LIN {X 0,Y 738.083,Z 977.53,A -85,B 0,C 180,E1 1734.319,E2 1734.319} C_VEL
LIN {X 0,Y 737.936,Z 977.53,A -85,B 0,C 180,E1 1739.532,E2 1739.532} C_VEL
LIN {X 0,Y 737.93,Z 977.53,A -85,B 0,C 180,E1 1743.677,E2 1743.677} C_VEL
LIN {X 0,Y 738.024,Z 977.53,A -85,B 0,C 180,E1 1748.027,E2 1748.027} C_VEL
LIN {X 0,Y 738.112,Z 977.53,A -85,B 0,C 180,E1 1752.652,E2 1752.652} C_VEL
LIN {X 0,Y 737.771,Z 977.53,A -85,B 0,C 180,E1 1757.348,E2 1757.348} C_VEL
LIN {X 0,Y 737.853,Z 977.53,A -85,B 0,C 180,E1 1761.985,E2 1761.985} C_VEL
LIN {X 0,Y 737.898,Z 977.53,A -85,B 0,C 180,E1 1766.342,E2 1766.342} C_VEL
LIN {X 0,Y 737.924,Z 977.53,A -85,B 0,C 180,E1 1770.487,E2 1770.487} C_VEL
LIN {X 0,Y 738.142,Z 977.53,A -85,B 0,C 180,E1 1774.599,E2 1774.599} C_VEL
LIN {X 0,Y 738.129,Z 977.53,A -85,B 0,C 180,E1 1778.326,E2 1778.326} C_VEL
LIN {X 0,Y 738.12,Z 977.53,A -85,B 0,C 180,E1 1783.308,E2 1783.308} C_VEL
LIN {X 0,Y 737.942,Z 977.53,A -85,B 0,C 180,E1 1788.161,E2 1788.161} C_VEL
LIN {X 0,Y 738.251,Z 977.53,A -85,B 0,C 180,E1 1792.935,E2 1792.935} C_VEL
LIN {X 0,Y 738.292,Z 977.708,A -85,B 0,C 180,E1 1797.418,E2 1797.418} C_VEL
LIN {X 0,Y 739.15,Z 1042.368,A -85,B 0,C 180,E1 1798.136,E2 1798.136} C_VEL
LIN {X 0,Y 738.978,Z 1071.102,A -85,B 0,C 180,E1 1798.907,E2 1798.907} C_VEL
LIN {X 0,Y 738.829,Z 1097.085,A -85,B 0,C 180,E1 1800.082,E2 1800.082} C_VEL
LIN {X 0,Y 738.695,Z 1119.698,A -85,B 0,C 180,E1 1801.624,E2 1801.624} C_VEL
LIN {X 0,Y 738.563,Z 1137.55,A -85,B 0,C 180,E1 1803.39,E2 1803.39} C_VEL
LIN {X 0,Y 738.525,Z 1151.255,A -85,B 0,C 180,E1 1805.451,E2 1805.451} C_VEL
LIN {X 0,Y 738.508,Z 1159.667,A -85,B 0,C 180,E1 1807.672,E2 1807.672} C_VEL
LIN {X 0,Y 738.433,Z 1162.462,A -85,B 0,C 180,E1 1809.919,E2 1809.919} C_VEL
LIN {X 0,Y 738.494,Z 1159.188,A -85,B 0,C 180,E1 1812.422,E2 1812.422} C_VEL
LIN {X 0,Y 738.524,Z 1150.902,A -85,B 0,C 180,E1 1814.527,E2 1814.527} C_VEL
LIN {X 0,Y 738.586,Z 1137.348,A -85,B 0,C 180,E1 1816.545,E2 1816.545} C_VEL
LIN {X 0,Y 738.661,Z 1118.397,A -85,B 0,C 180,E1 1818.391,E2 1818.391} C_VEL
LIN {X 0,Y 738.816,Z 1095.712,A -85,B 0,C 180,E1 1819.903,E2 1819.903} C_VEL
LIN {X 0,Y 738.997,Z 1069.193,A -85,B 0,C 180,E1 1821.071,E2 1821.071} C_VEL
LIN {X 0,Y 739.128,Z 1039.916,A -85,B 0,C 180,E1 1821.82,E2 1821.82} C_VEL
LIN {X 0,Y 738.331,Z 977.53,A -85,B 0,C 180,E1 1822.539,E2 1822.539} C_VEL
LIN {X 0,Y 738.05,Z 977.53,A -85,B 0,C 180,E1 1828.183,E2 1828.183} C_VEL
LIN {X 0,Y 737.952,Z 977.53,A -85,B 0,C 180,E1 1833.675,E2 1833.675} C_VEL
LIN {X 0,Y 737.897,Z 977.53,A -85,B 0,C 180,E1 1838.701,E2 1838.701} C_VEL
LIN {X 0,Y 738.199,Z 977.53,A -85,B 0,C 180,E1 1844.264,E2 1844.264} C_VEL
LIN {X 0,Y 738.006,Z 977.53,A -85,B 0,C 180,E1 1850.463,E2 1850.463} C_VEL
LIN {X 0,Y 737.986,Z 977.53,A -85,B 0,C 180,E1 1855.22,E2 1855.22} C_VEL
LIN {X 0,Y 737.948,Z 977.53,A -85,B 0,C 180,E1 1860.469,E2 1860.469} C_VEL
LIN {X 0,Y 738.116,Z 977.53,A -85,B 0,C 180,E1 1864.596,E2 1864.596} C_VEL
LIN {X 0,Y 738.118,Z 977.53,A -85,B 0,C 180,E1 1868.308,E2 1868.308} C_VEL
LIN {X 0,Y 738.114,Z 977.53,A -85,B 0,C 180,E1 1873.292,E2 1873.292} C_VEL
LIN {X 0,Y 737.966,Z 977.53,A -85,B 0,C 180,E1 1878.146,E2 1878.146} C_VEL
LIN {X 0,Y 738.261,Z 977.53,A -85,B 0,C 180,E1 1882.921,E2 1882.921} C_VEL
LIN {X 0,Y 738.268,Z 977.53,A -85,B 0,C 180,E1 1887.642,E2 1887.642} C_VEL
LIN {X 0,Y 738.112,Z 977.53,A -85,B 0,C 180,E1 1892.348,E2 1892.348} C_VEL
LIN {X 0,Y 738.101,Z 977.53,A -85,B 0,C 180,E1 1895.886,E2 1895.886} C_VEL
LIN {X 0,Y 738.049,Z 977.53,A -85,B 0,C 180,E1 1900.642,E2 1900.642} C_VEL
LIN {X 0,Y 738.137,Z 977.53,A -85,B 0,C 180,E1 1905.472,E2 1905.472} C_VEL
LIN {X 0,Y 738.142,Z 977.53,A -85,B 0,C 180,E1 1910.419,E2 1910.419} C_VEL
LIN {X 0,Y 737.968,Z 977.53,A -85,B 0,C 180,E1 1915.537,E2 1915.537} C_VEL
LIN {X 0,Y 737.941,Z 977.53,A -85,B 0,C 180,E1 1920.406,E2 1920.406} C_VEL
LIN {X 0,Y 737.901,Z 977.53,A -85,B 0,C 180,E1 1925.091,E2 1925.091} C_VEL
LIN {X 0,Y 737.805,Z 977.53,A -85,B 0,C 180,E1 1929.536,E2 1929.536} C_VEL
LIN {X 0,Y 738.181,Z 977.53,A -85,B 0,C 180,E1 1934.252,E2 1934.252} C_VEL
LIN {X 0,Y 738.006,Z 977.53,A -85,B 0,C 180,E1 1940.464,E2 1940.464} C_VEL
LIN {X 0,Y 737.961,Z 977.53,A -85,B 0,C 180,E1 1945.208,E2 1945.208} C_VEL
LIN {X 0,Y 737.934,Z 977.53,A -85,B 0,C 180,E1 1950.469,E2 1950.469} C_VEL
LIN {X 0,Y 738.209,Z 977.53,A -85,B 0,C 180,E1 1954.563,E2 1954.563} C_VEL
LIN {X 0,Y 738.21,Z 977.53,A -85,B 0,C 180,E1 1956.301,E2 1956.301} C_VEL
LIN {X 0,Y 740.647,Z 991.023,A -85,B 0,C 180,E1 1956.531,E2 1956.531} C_VEL
LIN {X 0,Y 740.707,Z 1032.457,A -85,B 0,C 180,E1 1957.203,E2 1957.203} C_VEL
LIN {X 0,Y 740.278,Z 1072.21,A -85,B 0,C 180,E1 1958.335,E2 1958.335} C_VEL
LIN {X 0,Y 739.819,Z 1109.026,A -85,B 0,C 180,E1 1959.882,E2 1959.882} C_VEL
LIN {X 0,Y 739.346,Z 1143.443,A -85,B 0,C 180,E1 1961.858,E2 1961.858} C_VEL
LIN {X 0,Y 738.974,Z 1173.471,A -85,B 0,C 180,E1 1964.135,E2 1964.135} C_VEL
LIN {X 0,Y 738.738,Z 1198.859,A -85,B 0,C 180,E1 1966.651,E2 1966.651} C_VEL
LIN {X 0,Y 738.54,Z 1219.45,A -85,B 0,C 180,E1 1969.352,E2 1969.352} C_VEL
LIN {X 0,Y 738.44,Z 1235.76,A -85,B 0,C 180,E1 1972.328,E2 1972.328} C_VEL
LIN {X 0,Y 738.388,Z 1246.269,A -85,B 0,C 180,E1 1975.284,E2 1975.284} C_VEL
LIN {X 0,Y 738.437,Z 1250.945,A -85,B 0,C 180,E1 1977.64,E2 1977.64} C_VEL
LIN {X 0,Y 738.33,Z 1252.496,A -85,B 0,C 180,E1 1979.992,E2 1979.992} C_VEL
LIN {X 0,Y 738.418,Z 1251.087,A -85,B 0,C 180,E1 1982.102,E2 1982.102} C_VEL
LIN {X 0,Y 735.908,Z 1249.732,A -85,B 0,C 180,E1 1983.098,E2 1983.098} C_VEL
LIN {X 0,Y 730.566,Z 1246.544,A -85,B 0,C 180,E1 1984.572,E2 1984.572} C_VEL
LIN {X 0,Y 730.486,Z 1246.099,A -85,B 0,C 180,E1 1984.742,E2 1984.742} C_VEL
LIN {X 0,Y 730.536,Z 1235.433,A -85,B 0,C 180,E1 1987.739,E2 1987.739} C_VEL
LIN {X 0,Y 730.659,Z 1219.999,A -85,B 0,C 180,E1 1990.59,E2 1990.59} C_VEL
LIN {X 0,Y 730.901,Z 1198.223,A -85,B 0,C 180,E1 1993.477,E2 1993.477} C_VEL
LIN {X 0,Y 731.297,Z 1171.96,A -85,B 0,C 180,E1 1996.078,E2 1996.078} C_VEL
LIN {X 0,Y 731.802,Z 1140.081,A -85,B 0,C 180,E1 1998.474,E2 1998.474} C_VEL
LIN {X 0,Y 732.31,Z 1104.123,A -85,B 0,C 180,E1 2000.483,E2 2000.483} C_VEL
LIN {X 0,Y 732.872,Z 1066.81,A -85,B 0,C 180,E1 2001.991,E2 2001.991} C_VEL
LIN {X 0,Y 733.297,Z 1027.462,A -85,B 0,C 180,E1 2003.056,E2 2003.056} C_VEL
LIN {X 0,Y 732.827,Z 985.525,A -85,B 0,C 180,E1 2003.701,E2 2003.701} C_VEL
LIN {X 0,Y 730.205,Z 977.53,A -85,B 0,C 180,E1 2003.916,E2 2003.916} C_VEL
LIN {X 0,Y 730.017,Z 977.53,A -85,B 0,C 180,E1 2009.346,E2 2009.346} C_VEL
LIN {X 0,Y 729.986,Z 977.53,A -85,B 0,C 180,E1 2014.072,E2 2014.072} C_VEL
LIN {X 0,Y 729.99,Z 977.53,A -85,B 0,C 180,E1 2018.499,E2 2018.499} C_VEL
LIN {X 0,Y 729.9,Z 977.53,A -85,B 0,C 180,E1 2023.406,E2 2023.406} C_VEL
LIN {X 0,Y 729.922,Z 977.53,A -85,B 0,C 180,E1 2028.379,E2 2028.379} C_VEL
LIN {X 0,Y 730.177,Z 977.53,A -85,B 0,C 180,E1 2033.008,E2 2033.008} C_VEL
LIN {X 0,Y 730.044,Z 977.53,A -85,B 0,C 180,E1 2037.347,E2 2037.347} C_VEL
LIN {X 0,Y 729.987,Z 977.53,A -85,B 0,C 180,E1 2042.834,E2 2042.834} C_VEL
LIN {X 0,Y 730.125,Z 977.53,A -85,B 0,C 180,E1 2045.43,E2 2045.43} C_VEL
LIN {X 0,Y 733.341,Z 989.383,A -85,B 0,C 180,E1 2045.682,E2 2045.682} C_VEL
LIN {X 0,Y 733.389,Z 1076.922,A -85,B 0,C 180,E1 2046.694,E2 2046.694} C_VEL
LIN {X 0,Y 733.015,Z 1118.546,A -85,B 0,C 180,E1 2047.697,E2 2047.697} C_VEL
LIN {X 0,Y 732.49,Z 1156.779,A -85,B 0,C 180,E1 2049.132,E2 2049.132} C_VEL
LIN {X 0,Y 731.917,Z 1191.997,A -85,B 0,C 180,E1 2050.976,E2 2050.976} C_VEL
LIN {X 0,Y 731.405,Z 1223.143,A -85,B 0,C 180,E1 2053.145,E2 2053.145} C_VEL
LIN {X 0,Y 730.936,Z 1250.193,A -85,B 0,C 180,E1 2055.601,E2 2055.601} C_VEL
LIN {X 0,Y 730.713,Z 1273.023,A -85,B 0,C 180,E1 2058.341,E2 2058.341} C_VEL
LIN {X 0,Y 730.516,Z 1289.835,A -85,B 0,C 180,E1 2061.056,E2 2061.056} C_VEL
LIN {X 0,Y 730.477,Z 1302.613,A -85,B 0,C 180,E1 2064.052,E2 2064.052} C_VEL
LIN {X 0,Y 730.456,Z 1308.949,A -85,B 0,C 180,E1 2066.438,E2 2066.438} C_VEL
LIN {X 0,Y 730.463,Z 1312.095,A -85,B 0,C 180,E1 2068.817,E2 2068.817} C_VEL
LIN {X 0,Y 730.436,Z 1312.086,A -85,B 0,C 180,E1 2071.194,E2 2071.194} C_VEL
LIN {X 0,Y 730.485,Z 1307.687,A -85,B 0,C 180,E1 2074.169,E2 2074.169} C_VEL
LIN {X 0,Y 730.59,Z 1296.916,A -85,B 0,C 180,E1 2077.454,E2 2077.454} C_VEL
LIN {X 0,Y 730.655,Z 1280.995,A -85,B 0,C 180,E1 2080.481,E2 2080.481} C_VEL
LIN {X 0,Y 730.926,Z 1259.819,A -85,B 0,C 180,E1 2083.34,E2 2083.34} C_VEL
LIN {X 0,Y 731.281,Z 1234.027,A -85,B 0,C 180,E1 2085.941,E2 2085.941} C_VEL
LIN {X 0,Y 731.699,Z 1203.965,A -85,B 0,C 180,E1 2088.259,E2 2088.259} C_VEL
LIN {X 0,Y 732.29,Z 1168.807,A -85,B 0,C 180,E1 2090.301,E2 2090.301} C_VEL
LIN {X 0,Y 732.865,Z 1129.891,A -85,B 0,C 180,E1 2091.933,E2 2091.933} C_VEL
LIN {X 0,Y 733.333,Z 1090.142,A -85,B 0,C 180,E1 2093.044,E2 2093.044} C_VEL
LIN {X 0,Y 733.53,Z 1051.079,A -85,B 0,C 180,E1 2093.664,E2 2093.664} C_VEL
LIN {X 0,Y 732.505,Z 984.943,A -85,B 0,C 180,E1 2094.395,E2 2094.395} C_VEL
LIN {X 0,Y 730.103,Z 977.53,A -85,B 0,C 180,E1 2094.599,E2 2094.599} C_VEL
LIN {X 0,Y 730.017,Z 977.53,A -85,B 0,C 180,E1 2099.884,E2 2099.884} C_VEL
LIN {X 0,Y 729.978,Z 977.53,A -85,B 0,C 180,E1 2104.094,E2 2104.094} C_VEL
LIN {X 0,Y 730.021,Z 977.53,A -85,B 0,C 180,E1 2108.52,E2 2108.52} C_VEL
LIN {X 0,Y 730.197,Z 977.53,A -85,B 0,C 180,E1 2113.442,E2 2113.442} C_VEL
LIN {X 0,Y 729.863,Z 977.53,A -85,B 0,C 180,E1 2118.385,E2 2118.385} C_VEL
LIN {X 0,Y 729.924,Z 977.53,A -85,B 0,C 180,E1 2123.001,E2 2123.001} C_VEL
LIN {X 0,Y 729.986,Z 977.53,A -85,B 0,C 180,E1 2127.352,E2 2127.352} C_VEL
LIN {X 0,Y 730.001,Z 977.53,A -85,B 0,C 180,E1 2131.497,E2 2131.497} C_VEL
LIN {X 0,Y 730.143,Z 977.53,A -85,B 0,C 180,E1 2135.955,E2 2135.955} C_VEL
LIN {X 0,Y 730.126,Z 977.53,A -85,B 0,C 180,E1 2140.618,E2 2140.618} C_VEL
LIN {X 0,Y 730.143,Z 977.53,A -85,B 0,C 180,E1 2145.59,E2 2145.59} C_VEL
LIN {X 0,Y 730.246,Z 977.53,A -85,B 0,C 180,E1 2150.454,E2 2150.454} C_VEL
LIN {X 0,Y 730.19,Z 977.53,A -85,B 0,C 180,E1 2155.248,E2 2155.248} C_VEL
LIN {X 0,Y 730.403,Z 977.53,A -85,B 0,C 180,E1 2157.259,E2 2157.259} C_VEL
LIN {X 0,Y 731.396,Z 1011.86,A -85,B 0,C 180,E1 2157.634,E2 2157.634} C_VEL
LIN {X 0,Y 731.367,Z 1047.602,A -85,B 0,C 180,E1 2158.116,E2 2158.116} C_VEL
LIN {X 0,Y 731.167,Z 1076.01,A -85,B 0,C 180,E1 2158.97,E2 2158.97} C_VEL
LIN {X 0,Y 730.977,Z 1101.516,A -85,B 0,C 180,E1 2160.231,E2 2160.231} C_VEL
LIN {X 0,Y 730.851,Z 1122.77,A -85,B 0,C 180,E1 2161.79,E2 2161.79} C_VEL
LIN {X 0,Y 730.706,Z 1140.681,A -85,B 0,C 180,E1 2163.724,E2 2163.724} C_VEL
LIN {X 0,Y 730.625,Z 1153.886,A -85,B 0,C 180,E1 2165.96,E2 2165.96} C_VEL
LIN {X 0,Y 730.594,Z 1159.901,A -85,B 0,C 180,E1 2167.755,E2 2167.755} C_VEL
LIN {X 0,Y 730.545,Z 1162.396,A -85,B 0,C 180,E1 2169.559,E2 2169.559} C_VEL
LIN {X 0,Y 730.576,Z 1160.301,A -85,B 0,C 180,E1 2171.978,E2 2171.978} C_VEL
LIN {X 0,Y 730.631,Z 1153.147,A -85,B 0,C 180,E1 2174.111,E2 2174.111} C_VEL
LIN {X 0,Y 730.75,Z 1140.113,A -85,B 0,C 180,E1 2176.263,E2 2176.263} C_VEL
LIN {X 0,Y 730.773,Z 1122.69,A -85,B 0,C 180,E1 2178.128,E2 2178.128} C_VEL
LIN {X 0,Y 730.961,Z 1099.874,A -85,B 0,C 180,E1 2179.778,E2 2179.778} C_VEL
LIN {X 0,Y 731.219,Z 1073.686,A -85,B 0,C 180,E1 2181.026,E2 2181.026} C_VEL
LIN {X 0,Y 731.393,Z 1044.893,A -85,B 0,C 180,E1 2181.849,E2 2181.849} C_VEL
LIN {X 0,Y 731.355,Z 996.33,A -85,B 0,C 180,E1 2182.43,E2 2182.43} C_VEL
LIN {X 0,Y 730.431,Z 977.53,A -85,B 0,C 180,E1 2182.686,E2 2182.686} C_VEL
LIN {X 0,Y 730.086,Z 977.53,A -85,B 0,C 180,E1 2188.519,E2 2188.519} C_VEL
LIN {X 0,Y 730.03,Z 977.53,A -85,B 0,C 180,E1 2193.866,E2 2193.866} C_VEL
LIN {X 0,Y 730.022,Z 977.53,A -85,B 0,C 180,E1 2198.518,E2 2198.518} C_VEL
LIN {X 0,Y 730.21,Z 977.53,A -85,B 0,C 180,E1 2203.416,E2 2203.416} C_VEL
LIN {X 0,Y 729.892,Z 977.53,A -85,B 0,C 180,E1 2208.368,E2 2208.368} C_VEL
LIN {X 0,Y 729.929,Z 977.53,A -85,B 0,C 180,E1 2212.979,E2 2212.979} C_VEL
LIN {X 0,Y 730,Z 977.53,A -85,B 0,C 180,E1 2217.331,E2 2217.331} C_VEL
LIN {X 0,Y 729.994,Z 977.53,A -85,B 0,C 180,E1 2221.477,E2 2221.477} C_VEL
LIN {X 0,Y 730.105,Z 977.53,A -85,B 0,C 180,E1 2225.954,E2 2225.954} C_VEL
LIN {X 0,Y 730.095,Z 977.53,A -85,B 0,C 180,E1 2230.6,E2 2230.6} C_VEL
LIN {X 0,Y 730.159,Z 977.53,A -85,B 0,C 180,E1 2235.574,E2 2235.574} C_VEL
LIN {X 0,Y 730.276,Z 977.53,A -85,B 0,C 180,E1 2240.439,E2 2240.439} C_VEL
LIN {X 0,Y 730.197,Z 977.53,A -85,B 0,C 180,E1 2245.233,E2 2245.233} C_VEL
LIN {X 0,Y 730.272,Z 977.53,A -85,B 0,C 180,E1 2249.994,E2 2249.994} C_VEL
LIN {X 0,Y 730.341,Z 977.53,A -85,B 0,C 180,E1 2255.189,E2 2255.189} C_VEL
LIN {X 0,Y 730.193,Z 977.53,A -85,B 0,C 180,E1 2259.55,E2 2259.55} C_VEL
LIN {X 0,Y 730.1,Z 977.53,A -85,B 0,C 180,E1 2264.416,E2 2264.416} C_VEL
LIN {X 0,Y 730.224,Z 977.53,A -85,B 0,C 180,E1 2269.385,E2 2269.385} C_VEL
LIN {X 0,Y 730.175,Z 977.53,A -85,B 0,C 180,E1 2274.516,E2 2274.516} C_VEL
LIN {X 0,Y 730.029,Z 977.53,A -85,B 0,C 180,E1 2279.871,E2 2279.871} C_VEL
LIN {X 0,Y 730.038,Z 977.53,A -85,B 0,C 180,E1 2284.077,E2 2284.077} C_VEL
LIN {X 0,Y 730.019,Z 977.53,A -85,B 0,C 180,E1 2288.506,E2 2288.506} C_VEL
LIN {X 0,Y 730.196,Z 977.53,A -85,B 0,C 180,E1 2293.418,E2 2293.418} C_VEL
LIN {X 0,Y 729.901,Z 977.53,A -85,B 0,C 180,E1 2298.365,E2 2298.365} C_VEL
LIN {X 0,Y 729.934,Z 977.53,A -85,B 0,C 180,E1 2302.981,E2 2302.981} C_VEL
LIN {X 0,Y 730.048,Z 977.53,A -85,B 0,C 180,E1 2308.308,E2 2308.308} C_VEL
LIN {X 0,Y 730.265,Z 977.53,A -85,B 0,C 180,E1 2314.162,E2 2314.162} C_VEL
LIN {X 0,Y 730.28,Z 977.53,A -85,B 0,C 180,E1 2316.026,E2 2316.026} C_VEL
LIN {X 0,Y 733.356,Z 991.134,A -85,B 0,C 180,E1 2316.286,E2 2316.286} C_VEL
LIN {X 0,Y 733.412,Z 1032.975,A -85,B 0,C 180,E1 2316.975,E2 2316.975} C_VEL
LIN {X 0,Y 732.849,Z 1072.247,A -85,B 0,C 180,E1 2318.106,E2 2318.106} C_VEL
LIN {X 0,Y 732.266,Z 1109.858,A -85,B 0,C 180,E1 2319.709,E2 2319.709} C_VEL
LIN {X 0,Y 731.728,Z 1143.436,A -85,B 0,C 180,E1 2321.663,E2 2321.663} C_VEL
LIN {X 0,Y 731.243,Z 1172.781,A -85,B 0,C 180,E1 2323.903,E2 2323.903} C_VEL
LIN {X 0,Y 730.948,Z 1198.856,A -85,B 0,C 180,E1 2326.507,E2 2326.507} C_VEL
LIN {X 0,Y 730.658,Z 1220.506,A -85,B 0,C 180,E1 2329.399,E2 2329.399} C_VEL
LIN {X 0,Y 730.575,Z 1235.758,A -85,B 0,C 180,E1 2332.244,E2 2332.244} C_VEL
LIN {X 0,Y 730.495,Z 1246.268,A -85,B 0,C 180,E1 2335.233,E2 2335.233} C_VEL
LIN {X 0,Y 730.53,Z 1250.945,A -85,B 0,C 180,E1 2337.614,E2 2337.614} C_VEL
LIN {X 0,Y 730.431,Z 1252.496,A -85,B 0,C 180,E1 2339.992,E2 2339.992} C_VEL
LIN {X 0,Y 730.54,Z 1250.84,A -85,B 0,C 180,E1 2342.369,E2 2342.369} C_VEL
LIN {X 0,Y 730.486,Z 1246.099,A -85,B 0,C 180,E1 2344.742,E2 2344.742} C_VEL
LIN {X 0,Y 729.255,Z 1244.28,A -85,B 0,C 180,E1 2345.407,E2 2345.407} C_VEL
LIN {X 0,Y 722.698,Z 1238.17,A -85,B 0,C 180,E1 2347.19,E2 2347.19} C_VEL
LIN {X 0,Y 722.63,Z 1237.478,A -85,B 0,C 180,E1 2347.355,E2 2347.355} C_VEL
LIN {X 0,Y 722.76,Z 1222.65,A -85,B 0,C 180,E1 2350.288,E2 2350.288} C_VEL
LIN {X 0,Y 723.06,Z 1200.886,A -85,B 0,C 180,E1 2353.317,E2 2353.317} C_VEL
LIN {X 0,Y 723.474,Z 1175.474,A -85,B 0,C 180,E1 2355.945,E2 2355.945} C_VEL
LIN {X 0,Y 724.038,Z 1145.817,A -85,B 0,C 180,E1 2358.284,E2 2358.284} C_VEL
LIN {X 0,Y 724.68,Z 1112.336,A -85,B 0,C 180,E1 2360.292,E2 2360.292} C_VEL
LIN {X 0,Y 725.376,Z 1076.129,A -85,B 0,C 180,E1 2361.894,E2 2361.894} C_VEL
LIN {X 0,Y 725.972,Z 1037.761,A -85,B 0,C 180,E1 2363.066,E2 2363.066} C_VEL
LIN {X 0,Y 726.328,Z 998.606,A -85,B 0,C 180,E1 2363.778,E2 2363.778} C_VEL
LIN {X 0,Y 725.571,Z 987.528,A -85,B 0,C 180,E1 2363.932,E2 2363.932} C_VEL
LIN {X 0,Y 722.21,Z 977.53,A -85,B 0,C 180,E1 2364.198,E2 2364.198} C_VEL
LIN {X 0,Y 722.128,Z 977.53,A -85,B 0,C 180,E1 2368.843,E2 2368.843} C_VEL
LIN {X 0,Y 722.164,Z 977.53,A -85,B 0,C 180,E1 2373.047,E2 2373.047} C_VEL
LIN {X 0,Y 722.222,Z 977.53,A -85,B 0,C 180,E1 2377.461,E2 2377.461} C_VEL
LIN {X 0,Y 721.978,Z 977.53,A -85,B 0,C 180,E1 2382.738,E2 2382.738} C_VEL
LIN {X 0,Y 721.984,Z 977.53,A -85,B 0,C 180,E1 2387.817,E2 2387.817} C_VEL
LIN {X 0,Y 722.273,Z 977.53,A -85,B 0,C 180,E1 2392.841,E2 2392.841} C_VEL
LIN {X 0,Y 722.131,Z 977.53,A -85,B 0,C 180,E1 2397.043,E2 2397.043} C_VEL
LIN {X 0,Y 722.063,Z 977.53,A -85,B 0,C 180,E1 2402.511,E2 2402.511} C_VEL
LIN {X 0,Y 722.19,Z 977.53,A -85,B 0,C 180,E1 2405.148,E2 2405.148} C_VEL
LIN {X 0,Y 726.184,Z 990.839,A -85,B 0,C 180,E1 2405.442,E2 2405.442} C_VEL
LIN {X 0,Y 726.11,Z 1076.424,A -85,B 0,C 180,E1 2406.438,E2 2406.438} C_VEL
LIN {X 0,Y 725.721,Z 1116.775,A -85,B 0,C 180,E1 2407.405,E2 2407.405} C_VEL
LIN {X 0,Y 725.077,Z 1154.731,A -85,B 0,C 180,E1 2408.815,E2 2408.815} C_VEL
LIN {X 0,Y 724.352,Z 1190.713,A -85,B 0,C 180,E1 2410.69,E2 2410.69} C_VEL
LIN {X 0,Y 723.689,Z 1223.143,A -85,B 0,C 180,E1 2412.96,E2 2412.96} C_VEL
LIN {X 0,Y 723.145,Z 1250.198,A -85,B 0,C 180,E1 2415.443,E2 2415.443} C_VEL
LIN {X 0,Y 722.856,Z 1273.021,A -85,B 0,C 180,E1 2418.212,E2 2418.212} C_VEL
LIN {X 0,Y 722.648,Z 1289.839,A -85,B 0,C 180,E1 2420.958,E2 2420.958} C_VEL
LIN {X 0,Y 722.578,Z 1302.611,A -85,B 0,C 180,E1 2423.987,E2 2423.987} C_VEL
LIN {X 0,Y 722.56,Z 1308.952,A -85,B 0,C 180,E1 2426.399,E2 2426.399} C_VEL
LIN {X 0,Y 722.59,Z 1312.098,A -85,B 0,C 180,E1 2428.804,E2 2428.804} C_VEL
LIN {X 0,Y 722.565,Z 1312.089,A -85,B 0,C 180,E1 2431.207,E2 2431.207} C_VEL
LIN {X 0,Y 722.606,Z 1307.683,A -85,B 0,C 180,E1 2434.214,E2 2434.214} C_VEL
LIN {X 0,Y 722.705,Z 1296.919,A -85,B 0,C 180,E1 2437.535,E2 2437.535} C_VEL
LIN {X 0,Y 722.794,Z 1280.941,A -85,B 0,C 180,E1 2440.604,E2 2440.604} C_VEL
LIN {X 0,Y 723.113,Z 1259.824,A -85,B 0,C 180,E1 2443.487,E2 2443.487} C_VEL
LIN {X 0,Y 723.523,Z 1234.026,A -85,B 0,C 180,E1 2446.116,E2 2446.116} C_VEL
LIN {X 0,Y 724.111,Z 1203.971,A -85,B 0,C 180,E1 2448.457,E2 2448.457} C_VEL
LIN {X 0,Y 724.744,Z 1170.082,A -85,B 0,C 180,E1 2450.456,E2 2450.456} C_VEL
LIN {X 0,Y 725.46,Z 1132.101,A -85,B 0,C 180,E1 2452.09,E2 2452.09} C_VEL
LIN {X 0,Y 726,Z 1092.6,A -85,B 0,C 180,E1 2453.237,E2 2453.237} C_VEL
LIN {X 0,Y 726.298,Z 1051.079,A -85,B 0,C 180,E1 2453.914,E2 2453.914} C_VEL
LIN {X 0,Y 725.421,Z 987.329,A -85,B 0,C 180,E1 2454.623,E2 2454.623} C_VEL
LIN {X 0,Y 722.163,Z 977.53,A -85,B 0,C 180,E1 2454.911,E2 2454.911} C_VEL
LIN {X 0,Y 722.082,Z 977.53,A -85,B 0,C 180,E1 2460.247,E2 2460.247} C_VEL
LIN {X 0,Y 722.054,Z 977.53,A -85,B 0,C 180,E1 2465.096,E2 2465.096} C_VEL
LIN {X 0,Y 722.025,Z 977.53,A -85,B 0,C 180,E1 2469.081,E2 2469.081} C_VEL
LIN {X 0,Y 722.248,Z 977.53,A -85,B 0,C 180,E1 2474.514,E2 2474.514} C_VEL
LIN {X 0,Y 722.021,Z 977.53,A -85,B 0,C 180,E1 2479.432,E2 2479.432} C_VEL
LIN {X 0,Y 722.058,Z 977.53,A -85,B 0,C 180,E1 2484.029,E2 2484.029} C_VEL
LIN {X 0,Y 722.162,Z 977.53,A -85,B 0,C 180,E1 2489.358,E2 2489.358} C_VEL
LIN {X 0,Y 722.259,Z 977.53,A -85,B 0,C 180,E1 2494.451,E2 2494.451} C_VEL
LIN {X 0,Y 722.204,Z 977.53,A -85,B 0,C 180,E1 2499.115,E2 2499.115} C_VEL
LIN {X 0,Y 722.24,Z 977.53,A -85,B 0,C 180,E1 2504.183,E2 2504.183} C_VEL
LIN {X 0,Y 722.368,Z 977.53,A -85,B 0,C 180,E1 2509.128,E2 2509.128} C_VEL
LIN {X 0,Y 722.425,Z 977.53,A -85,B 0,C 180,E1 2513.989,E2 2513.989} C_VEL
LIN {X 0,Y 722.528,Z 977.782,A -85,B 0,C 180,E1 2517.14,E2 2517.14} C_VEL
LIN {X 0,Y 723.657,Z 1006.321,A -85,B 0,C 180,E1 2517.445,E2 2517.445} C_VEL
LIN {X 0,Y 723.664,Z 1045.533,A -85,B 0,C 180,E1 2517.946,E2 2517.946} C_VEL
LIN {X 0,Y 723.442,Z 1073.862,A -85,B 0,C 180,E1 2518.771,E2 2518.771} C_VEL
LIN {X 0,Y 723.235,Z 1099.582,A -85,B 0,C 180,E1 2520.009,E2 2520.009} C_VEL
LIN {X 0,Y 723.012,Z 1122.309,A -85,B 0,C 180,E1 2521.66,E2 2521.66} C_VEL
LIN {X 0,Y 722.81,Z 1140.367,A -85,B 0,C 180,E1 2523.614,E2 2523.614} C_VEL
LIN {X 0,Y 722.733,Z 1153.07,A -85,B 0,C 180,E1 2525.739,E2 2525.739} C_VEL
LIN {X 0,Y 722.681,Z 1160.133,A -85,B 0,C 180,E1 2527.841,E2 2527.841} C_VEL
LIN {X 0,Y 722.63,Z 1162.436,A -85,B 0,C 180,E1 2529.726,E2 2529.726} C_VEL
LIN {X 0,Y 722.687,Z 1160.041,A -85,B 0,C 180,E1 2532.11,E2 2532.11} C_VEL
LIN {X 0,Y 722.736,Z 1152.618,A -85,B 0,C 180,E1 2534.269,E2 2534.269} C_VEL
LIN {X 0,Y 722.838,Z 1139.271,A -85,B 0,C 180,E1 2536.446,E2 2536.446} C_VEL
LIN {X 0,Y 722.96,Z 1121.386,A -85,B 0,C 180,E1 2538.331,E2 2538.331} C_VEL
LIN {X 0,Y 723.135,Z 1099.385,A -85,B 0,C 180,E1 2539.914,E2 2539.914} C_VEL
LIN {X 0,Y 723.476,Z 1073.818,A -85,B 0,C 180,E1 2541.14,E2 2541.14} C_VEL
LIN {X 0,Y 723.657,Z 1044.632,A -85,B 0,C 180,E1 2541.983,E2 2541.983} C_VEL
LIN {X 0,Y 723.632,Z 993.741,A -85,B 0,C 180,E1 2542.591,E2 2542.591} C_VEL
LIN {X 0,Y 722.512,Z 977.53,A -85,B 0,C 180,E1 2542.822,E2 2542.822} C_VEL
LIN {X 0,Y 722.152,Z 977.53,A -85,B 0,C 180,E1 2548.193,E2 2548.193} C_VEL
LIN {X 0,Y 722.173,Z 977.53,A -85,B 0,C 180,E1 2553.067,E2 2553.067} C_VEL
LIN {X 0,Y 722.217,Z 977.53,A -85,B 0,C 180,E1 2557.482,E2 2557.482} C_VEL
LIN {X 0,Y 722.225,Z 977.53,A -85,B 0,C 180,E1 2562.742,E2 2562.742} C_VEL
LIN {X 0,Y 721.978,Z 977.53,A -85,B 0,C 180,E1 2567.276,E2 2567.276} C_VEL
LIN {X 0,Y 722.016,Z 977.53,A -85,B 0,C 180,E1 2572.504,E2 2572.504} C_VEL
LIN {X 0,Y 722.083,Z 977.53,A -85,B 0,C 180,E1 2577.081,E2 2577.081} C_VEL
LIN {X 0,Y 722.096,Z 977.53,A -85,B 0,C 180,E1 2581.81,E2 2581.81} C_VEL
LIN {X 0,Y 722.245,Z 977.53,A -85,B 0,C 180,E1 2586.502,E2 2586.502} C_VEL
LIN {X 0,Y 722.263,Z 977.53,A -85,B 0,C 180,E1 2591.652,E2 2591.652} C_VEL
LIN {X 0,Y 722.154,Z 977.53,A -85,B 0,C 180,E1 2596.65,E2 2596.65} C_VEL
LIN {X 0,Y 722.373,Z 977.53,A -85,B 0,C 180,E1 2600.372,E2 2600.372} C_VEL
LIN {X 0,Y 722.319,Z 977.53,A -85,B 0,C 180,E1 2605.181,E2 2605.181} C_VEL
LIN {X 0,Y 722.381,Z 977.53,A -85,B 0,C 180,E1 2609.994,E2 2609.994} C_VEL
LIN {X 0,Y 722.555,Z 977.53,A -85,B 0,C 180,E1 2614.806,E2 2614.806} C_VEL
LIN {X 0,Y 722.277,Z 977.53,A -85,B 0,C 180,E1 2619.656,E2 2619.656} C_VEL
LIN {X 0,Y 722.199,Z 977.53,A -85,B 0,C 180,E1 2624.577,E2 2624.577} C_VEL
LIN {X 0,Y 722.293,Z 977.53,A -85,B 0,C 180,E1 2629.606,E2 2629.606} C_VEL
LIN {X 0,Y 722.211,Z 977.53,A -85,B 0,C 180,E1 2634.804,E2 2634.804} C_VEL
LIN {X 0,Y 722.152,Z 977.53,A -85,B 0,C 180,E1 2638.849,E2 2638.849} C_VEL
LIN {X 0,Y 722.192,Z 977.53,A -85,B 0,C 180,E1 2643.053,E2 2643.053} C_VEL
LIN {X 0,Y 722.205,Z 977.53,A -85,B 0,C 180,E1 2647.47,E2 2647.47} C_VEL
LIN {X 0,Y 722.221,Z 977.53,A -85,B 0,C 180,E1 2652.745,E2 2652.745} C_VEL
LIN {X 0,Y 721.979,Z 977.53,A -85,B 0,C 180,E1 2657.804,E2 2657.804} C_VEL
LIN {X 0,Y 722.053,Z 977.53,A -85,B 0,C 180,E1 2662.878,E2 2662.878} C_VEL
LIN {X 0,Y 722.165,Z 977.53,A -85,B 0,C 180,E1 2668.356,E2 2668.356} C_VEL
LIN {X 0,Y 722.337,Z 977.53,A -85,B 0,C 180,E1 2673.857,E2 2673.857} C_VEL
LIN {X 0,Y 722.378,Z 977.53,A -85,B 0,C 180,E1 2675.758,E2 2675.758} C_VEL
LIN {X 0,Y 726.151,Z 992.19,A -85,B 0,C 180,E1 2676.047,E2 2676.047} C_VEL
LIN {X 0,Y 726.103,Z 1033.812,A -85,B 0,C 180,E1 2676.751,E2 2676.751} C_VEL
LIN {X 0,Y 725.443,Z 1073.252,A -85,B 0,C 180,E1 2677.909,E2 2677.909} C_VEL
LIN {X 0,Y 724.747,Z 1109.651,A -85,B 0,C 180,E1 2679.479,E2 2679.479} C_VEL
LIN {X 0,Y 724.107,Z 1143.428,A -85,B 0,C 180,E1 2681.463,E2 2681.463} C_VEL
LIN {X 0,Y 723.51,Z 1172.777,A -85,B 0,C 180,E1 2683.726,E2 2683.726} C_VEL
LIN {X 0,Y 723.145,Z 1198.854,A -85,B 0,C 180,E1 2686.358,E2 2686.358} C_VEL
LIN {X 0,Y 722.831,Z 1219.446,A -85,B 0,C 180,E1 2689.118,E2 2689.118} C_VEL
LIN {X 0,Y 722.718,Z 1235.757,A -85,B 0,C 180,E1 2692.16,E2 2692.16} C_VEL
LIN {X 0,Y 722.6,Z 1246.267,A -85,B 0,C 180,E1 2695.18,E2 2695.18} C_VEL
LIN {X 0,Y 722.646,Z 1250.944,A -85,B 0,C 180,E1 2697.588,E2 2697.588} C_VEL
LIN {X 0,Y 722.559,Z 1252.496,A -85,B 0,C 180,E1 2699.991,E2 2699.991} C_VEL
LIN {X 0,Y 722.659,Z 1250.841,A -85,B 0,C 180,E1 2702.395,E2 2702.395} C_VEL
LIN {X 0,Y 722.697,Z 1243.969,A -85,B 0,C 180,E1 2705.542,E2 2705.542} C_VEL
LIN {X 0,Y 722.63,Z 1237.478,A -85,B 0,C 180,E1 2707.355,E2 2707.355} C_VEL
LIN {X 0,Y 721.466,Z 1234.687,A -85,B 0,C 180,E1 2708.007,E2 2708.007} C_VEL
LIN {X 0,Y 714.966,Z 1226.341,A -85,B 0,C 180,E1 2709.751,E2 2709.751} C_VEL
LIN {X 0,Y 714.873,Z 1225.435,A -85,B 0,C 180,E1 2709.912,E2 2709.912} C_VEL
LIN {X 0,Y 715.12,Z 1205.968,A -85,B 0,C 180,E1 2712.831,E2 2712.831} C_VEL
LIN {X 0,Y 715.657,Z 1181.037,A -85,B 0,C 180,E1 2715.599,E2 2715.599} C_VEL
LIN {X 0,Y 716.283,Z 1151.507,A -85,B 0,C 180,E1 2718.084,E2 2718.084} C_VEL
LIN {X 0,Y 717.106,Z 1116.528,A -85,B 0,C 180,E1 2720.293,E2 2720.293} C_VEL
LIN {X 0,Y 717.929,Z 1080.765,A -85,B 0,C 180,E1 2721.954,E2 2721.954} C_VEL
LIN {X 0,Y 718.669,Z 1042.546,A -85,B 0,C 180,E1 2723.192,E2 2723.192} C_VEL
LIN {X 0,Y 719.084,Z 1003.949,A -85,B 0,C 180,E1 2723.962,E2 2723.962} C_VEL
LIN {X 0,Y 718.271,Z 989.117,A -85,B 0,C 180,E1 2724.175,E2 2724.175} C_VEL
LIN {X 0,Y 714.229,Z 977.53,A -85,B 0,C 180,E1 2724.498,E2 2724.498} C_VEL
LIN {X 0,Y 714.15,Z 977.53,A -85,B 0,C 180,E1 2729.562,E2 2729.562} C_VEL
LIN {X 0,Y 714.138,Z 977.53,A -85,B 0,C 180,E1 2734.167,E2 2734.167} C_VEL
LIN {X 0,Y 714.149,Z 977.53,A -85,B 0,C 180,E1 2738.283,E2 2738.283} C_VEL
LIN {X 0,Y 714.029,Z 977.53,A -85,B 0,C 180,E1 2743.828,E2 2743.828} C_VEL
LIN {X 0,Y 714.022,Z 977.53,A -85,B 0,C 180,E1 2748.87,E2 2748.87} C_VEL
LIN {X 0,Y 714.334,Z 977.53,A -85,B 0,C 180,E1 2753.689,E2 2753.689} C_VEL
LIN {X 0,Y 714.195,Z 977.53,A -85,B 0,C 180,E1 2758.038,E2 2758.038} C_VEL
LIN {X 0,Y 714.1,Z 977.53,A -85,B 0,C 180,E1 2762.993,E2 2762.993} C_VEL
LIN {X 0,Y 714.228,Z 977.53,A -85,B 0,C 180,E1 2764.855,E2 2764.855} C_VEL
LIN {X 0,Y 719.074,Z 994.112,A -85,B 0,C 180,E1 2765.218,E2 2765.218} C_VEL
LIN {X 0,Y 718.874,Z 1076.66,A -85,B 0,C 180,E1 2766.191,E2 2766.191} C_VEL
LIN {X 0,Y 718.355,Z 1117.879,A -85,B 0,C 180,E1 2767.196,E2 2767.196} C_VEL
LIN {X 0,Y 717.584,Z 1156.06,A -85,B 0,C 180,E1 2768.645,E2 2768.645} C_VEL
LIN {X 0,Y 716.737,Z 1191.993,A -85,B 0,C 180,E1 2770.557,E2 2770.557} C_VEL
LIN {X 0,Y 716.011,Z 1223.138,A -85,B 0,C 180,E1 2772.772,E2 2772.772} C_VEL
LIN {X 0,Y 715.355,Z 1250.203,A -85,B 0,C 180,E1 2775.281,E2 2775.281} C_VEL
LIN {X 0,Y 715.014,Z 1273.019,A -85,B 0,C 180,E1 2778.081,E2 2778.081} C_VEL
LIN {X 0,Y 714.773,Z 1289.844,A -85,B 0,C 180,E1 2780.857,E2 2780.857} C_VEL
LIN {X 0,Y 714.711,Z 1302.609,A -85,B 0,C 180,E1 2783.921,E2 2783.921} C_VEL
LIN {X 0,Y 714.662,Z 1308.956,A -85,B 0,C 180,E1 2786.359,E2 2786.359} C_VEL
LIN {X 0,Y 714.689,Z 1312.1,A -85,B 0,C 180,E1 2788.791,E2 2788.791} C_VEL
LIN {X 0,Y 714.664,Z 1312.091,A -85,B 0,C 180,E1 2791.221,E2 2791.221} C_VEL
LIN {X 0,Y 714.703,Z 1307.679,A -85,B 0,C 180,E1 2794.261,E2 2794.261} C_VEL
LIN {X 0,Y 714.839,Z 1296.923,A -85,B 0,C 180,E1 2797.619,E2 2797.619} C_VEL
LIN {X 0,Y 714.933,Z 1281.115,A -85,B 0,C 180,E1 2800.693,E2 2800.693} C_VEL
LIN {X 0,Y 715.315,Z 1259.828,A -85,B 0,C 180,E1 2803.636,E2 2803.636} C_VEL
LIN {X 0,Y 715.812,Z 1234.024,A -85,B 0,C 180,E1 2806.295,E2 2806.295} C_VEL
LIN {X 0,Y 716.494,Z 1203.978,A -85,B 0,C 180,E1 2808.661,E2 2808.661} C_VEL
LIN {X 0,Y 717.268,Z 1169.137,A -85,B 0,C 180,E1 2810.729,E2 2810.729} C_VEL
LIN {X 0,Y 718.081,Z 1132.107,A -85,B 0,C 180,E1 2812.329,E2 2812.329} C_VEL
LIN {X 0,Y 718.752,Z 1092.599,A -85,B 0,C 180,E1 2813.485,E2 2813.485} C_VEL
LIN {X 0,Y 719.097,Z 1052.802,A -85,B 0,C 180,E1 2814.15,E2 2814.15} C_VEL
LIN {X 0,Y 718.021,Z 988.582,A -85,B 0,C 180,E1 2814.881,E2 2814.881} C_VEL
LIN {X 0,Y 714.217,Z 977.53,A -85,B 0,C 180,E1 2815.2,E2 2815.2} C_VEL
LIN {X 0,Y 714.201,Z 977.53,A -85,B 0,C 180,E1 2820.616,E2 2820.616} C_VEL
LIN {X 0,Y 714.159,Z 977.53,A -85,B 0,C 180,E1 2824.958,E2 2824.958} C_VEL
LIN {X 0,Y 714.078,Z 977.53,A -85,B 0,C 180,E1 2829.546,E2 2829.546} C_VEL
LIN {X 0,Y 714.347,Z 977.53,A -85,B 0,C 180,E1 2834.434,E2 2834.434} C_VEL
LIN {X 0,Y 714.085,Z 977.53,A -85,B 0,C 180,E1 2839.818,E2 2839.818} C_VEL
LIN {X 0,Y 714.166,Z 977.53,A -85,B 0,C 180,E1 2845.065,E2 2845.065} C_VEL
LIN {X 0,Y 714.258,Z 977.53,A -85,B 0,C 180,E1 2849.407,E2 2849.407} C_VEL
LIN {X 0,Y 714.326,Z 977.53,A -85,B 0,C 180,E1 2854.91,E2 2854.91} C_VEL
LIN {X 0,Y 714.308,Z 977.53,A -85,B 0,C 180,E1 2858.982,E2 2858.982} C_VEL
LIN {X 0,Y 714.33,Z 977.53,A -85,B 0,C 180,E1 2864.004,E2 2864.004} C_VEL
LIN {X 0,Y 714.427,Z 977.53,A -85,B 0,C 180,E1 2869.006,E2 2869.006} C_VEL
LIN {X 0,Y 714.538,Z 977.53,A -85,B 0,C 180,E1 2873.923,E2 2873.923} C_VEL
LIN {X 0,Y 714.604,Z 977.53,A -85,B 0,C 180,E1 2876.97,E2 2876.97} C_VEL
LIN {X 0,Y 715.975,Z 995.914,A -85,B 0,C 180,E1 2877.204,E2 2877.204} C_VEL
LIN {X 0,Y 715.984,Z 1043.455,A -85,B 0,C 180,E1 2877.773,E2 2877.773} C_VEL
LIN {X 0,Y 715.705,Z 1072.695,A -85,B 0,C 180,E1 2878.606,E2 2878.606} C_VEL
LIN {X 0,Y 715.42,Z 1098.833,A -85,B 0,C 180,E1 2879.857,E2 2879.857} C_VEL
LIN {X 0,Y 715.182,Z 1121.84,A -85,B 0,C 180,E1 2881.526,E2 2881.526} C_VEL
LIN {X 0,Y 714.95,Z 1140.049,A -85,B 0,C 180,E1 2883.502,E2 2883.502} C_VEL
LIN {X 0,Y 714.859,Z 1153.483,A -85,B 0,C 180,E1 2885.786,E2 2885.786} C_VEL
LIN {X 0,Y 714.797,Z 1160.364,A -85,B 0,C 180,E1 2887.928,E2 2887.928} C_VEL
LIN {X 0,Y 714.75,Z 1162.424,A -85,B 0,C 180,E1 2889.772,E2 2889.772} C_VEL
LIN {X 0,Y 714.801,Z 1159.78,A -85,B 0,C 180,E1 2892.246,E2 2892.246} C_VEL
LIN {X 0,Y 714.853,Z 1152.09,A -85,B 0,C 180,E1 2894.429,E2 2894.429} C_VEL
LIN {X 0,Y 715,Z 1138.403,A -85,B 0,C 180,E1 2896.632,E2 2896.632} C_VEL
LIN {X 0,Y 715.159,Z 1120.026,A -85,B 0,C 180,E1 2898.538,E2 2898.538} C_VEL
LIN {X 0,Y 715.361,Z 1097.302,A -85,B 0,C 180,E1 2900.14,E2 2900.14} C_VEL
LIN {X 0,Y 715.724,Z 1070.17,A -85,B 0,C 180,E1 2901.398,E2 2901.398} C_VEL
LIN {X 0,Y 715.976,Z 1042.747,A -85,B 0,C 180,E1 2902.152,E2 2902.152} C_VEL
LIN {X 0,Y 715.155,Z 980.773,A -85,B 0,C 180,E1 2902.874,E2 2902.874} C_VEL
LIN {X 0,Y 714.611,Z 977.53,A -85,B 0,C 180,E1 2902.942,E2 2902.942} C_VEL
LIN {X 0,Y 714.246,Z 977.53,A -85,B 0,C 180,E1 2907.828,E2 2907.828} C_VEL
LIN {X 0,Y 714.242,Z 977.53,A -85,B 0,C 180,E1 2912.037,E2 2912.037} C_VEL
LIN {X 0,Y 714.24,Z 977.53,A -85,B 0,C 180,E1 2916.449,E2 2916.449} C_VEL
LIN {X 0,Y 714.236,Z 977.53,A -85,B 0,C 180,E1 2922.044,E2 2922.044} C_VEL
LIN {X 0,Y 714.188,Z 977.53,A -85,B 0,C 180,E1 2926.173,E2 2926.173} C_VEL
LIN {X 0,Y 714.108,Z 977.53,A -85,B 0,C 180,E1 2931.735,E2 2931.735} C_VEL
LIN {X 0,Y 714.12,Z 977.53,A -85,B 0,C 180,E1 2936.511,E2 2936.511} C_VEL
LIN {X 0,Y 714.171,Z 977.53,A -85,B 0,C 180,E1 2940.785,E2 2940.785} C_VEL
LIN {X 0,Y 714.288,Z 977.53,A -85,B 0,C 180,E1 2945.815,E2 2945.815} C_VEL
LIN {X 0,Y 714.27,Z 977.53,A -85,B 0,C 180,E1 2950.152,E2 2950.152} C_VEL
LIN {X 0,Y 714.359,Z 977.53,A -85,B 0,C 180,E1 2953.987,E2 2953.987} C_VEL
LIN {X 0,Y 714.488,Z 977.53,A -85,B 0,C 180,E1 2958.991,E2 2958.991} C_VEL
LIN {X 0,Y 714.531,Z 977.53,A -85,B 0,C 180,E1 2963.908,E2 2963.908} C_VEL
LIN {X 0,Y 714.416,Z 977.53,A -85,B 0,C 180,E1 2968.779,E2 2968.779} C_VEL
LIN {X 0,Y 714.408,Z 977.53,A -85,B 0,C 180,E1 2972.426,E2 2972.426} C_VEL
LIN {X 0,Y 714.382,Z 977.53,A -85,B 0,C 180,E1 2976.082,E2 2976.082} C_VEL
LIN {X 0,Y 714.335,Z 977.53,A -85,B 0,C 180,E1 2981,E2 2981} C_VEL
LIN {X 0,Y 714.422,Z 977.53,A -85,B 0,C 180,E1 2985.999,E2 2985.999} C_VEL
LIN {X 0,Y 714.329,Z 977.53,A -85,B 0,C 180,E1 2991.132,E2 2991.132} C_VEL
LIN {X 0,Y 714.275,Z 977.53,A -85,B 0,C 180,E1 2995.099,E2 2995.099} C_VEL
LIN {X 0,Y 714.17,Z 977.53,A -85,B 0,C 180,E1 2999.547,E2 2999.547} C_VEL
LIN {X 0,Y 714.179,Z 977.53,A -85,B 0,C 180,E1 3004.156,E2 3004.156} C_VEL
LIN {X 0,Y 714.17,Z 977.53,A -85,B 0,C 180,E1 3008.271,E2 3008.271} C_VEL
LIN {X 0,Y 714.369,Z 977.53,A -85,B 0,C 180,E1 3013.842,E2 3013.842} C_VEL
LIN {X 0,Y 714.103,Z 977.53,A -85,B 0,C 180,E1 3018.863,E2 3018.863} C_VEL
LIN {X 0,Y 714.149,Z 977.53,A -85,B 0,C 180,E1 3023.724,E2 3023.724} C_VEL
LIN {X 0,Y 714.266,Z 977.53,A -85,B 0,C 180,E1 3029.387,E2 3029.387} C_VEL
LIN {X 0,Y 714.405,Z 977.53,A -85,B 0,C 180,E1 3034.893,E2 3034.893} C_VEL
LIN {X 0,Y 714.452,Z 977.53,A -85,B 0,C 180,E1 3035.469,E2 3035.469} C_VEL
LIN {X 0,Y 718.88,Z 992.393,A -85,B 0,C 180,E1 3035.792,E2 3035.792} C_VEL
LIN {X 0,Y 718.815,Z 1033.8,A -85,B 0,C 180,E1 3036.501,E2 3036.501} C_VEL
LIN {X 0,Y 718.046,Z 1073.242,A -85,B 0,C 180,E1 3037.669,E2 3037.669} C_VEL
LIN {X 0,Y 717.259,Z 1109.927,A -85,B 0,C 180,E1 3039.27,E2 3039.27} C_VEL
LIN {X 0,Y 716.497,Z 1143.421,A -85,B 0,C 180,E1 3041.258,E2 3041.258} C_VEL
LIN {X 0,Y 715.796,Z 1172.773,A -85,B 0,C 180,E1 3043.546,E2 3043.546} C_VEL
LIN {X 0,Y 715.33,Z 1198.852,A -85,B 0,C 180,E1 3046.206,E2 3046.206} C_VEL
LIN {X 0,Y 714.972,Z 1219.444,A -85,B 0,C 180,E1 3048.997,E2 3048.997} C_VEL
LIN {X 0,Y 714.837,Z 1235.756,A -85,B 0,C 180,E1 3052.073,E2 3052.073} C_VEL
LIN {X 0,Y 714.708,Z 1246.266,A -85,B 0,C 180,E1 3055.127,E2 3055.127} C_VEL
LIN {X 0,Y 714.74,Z 1250.944,A -85,B 0,C 180,E1 3057.562,E2 3057.562} C_VEL
LIN {X 0,Y 714.659,Z 1252.497,A -85,B 0,C 180,E1 3059.991,E2 3059.991} C_VEL
LIN {X 0,Y 714.756,Z 1250.842,A -85,B 0,C 180,E1 3062.421,E2 3062.421} C_VEL
LIN {X 0,Y 714.791,Z 1244.409,A -85,B 0,C 180,E1 3065.464,E2 3065.464} C_VEL
LIN {X 0,Y 714.796,Z 1232.685,A -85,B 0,C 180,E1 3068.524,E2 3068.524} C_VEL
LIN {X 0,Y 714.873,Z 1225.435,A -85,B 0,C 180,E1 3069.912,E2 3069.912} C_VEL
LIN {X 0,Y 711.042,Z 1218.272,A -85,B 0,C 180,E1 3071.162,E2 3071.162} C_VEL
LIN {X 0,Y 707.254,Z 1210.348,A -85,B 0,C 180,E1 3072.393,E2 3072.393} C_VEL
LIN {X 0,Y 707.76,Z 1185.28,A -85,B 0,C 180,E1 3075.355,E2 3075.355} C_VEL
LIN {X 0,Y 708.44,Z 1156.801,A -85,B 0,C 180,E1 3077.884,E2 3077.884} C_VEL
LIN {X 0,Y 709.397,Z 1124.803,A -85,B 0,C 180,E1 3080.045,E2 3080.045} C_VEL
LIN {X 0,Y 710.301,Z 1089.409,A -85,B 0,C 180,E1 3081.837,E2 3081.837} C_VEL
LIN {X 0,Y 711.149,Z 1052.349,A -85,B 0,C 180,E1 3083.173,E2 3083.173} C_VEL
LIN {X 0,Y 711.745,Z 1013.462,A -85,B 0,C 180,E1 3084.073,E2 3084.073} C_VEL
LIN {X 0,Y 710.982,Z 991.008,A -85,B 0,C 180,E1 3084.419,E2 3084.419} C_VEL
LIN {X 0,Y 706.271,Z 977.53,A -85,B 0,C 180,E1 3084.786,E2 3084.786} C_VEL
LIN {X 0,Y 706.251,Z 977.53,A -85,B 0,C 180,E1 3089.555,E2 3089.555} C_VEL
LIN {X 0,Y 706.243,Z 977.53,A -85,B 0,C 180,E1 3093.891,E2 3093.891} C_VEL
LIN {X 0,Y 706.209,Z 977.53,A -85,B 0,C 180,E1 3098.463,E2 3098.463} C_VEL
LIN {X 0,Y 706.132,Z 977.53,A -85,B 0,C 180,E1 3103.349,E2 3103.349} C_VEL
LIN {X 0,Y 706.129,Z 977.53,A -85,B 0,C 180,E1 3108.661,E2 3108.661} C_VEL
LIN {X 0,Y 706.341,Z 977.53,A -85,B 0,C 180,E1 3113.09,E2 3113.09} C_VEL
LIN {X 0,Y 706.247,Z 977.53,A -85,B 0,C 180,E1 3117.569,E2 3117.569} C_VEL
LIN {X 0,Y 706.229,Z 977.53,A -85,B 0,C 180,E1 3121.841,E2 3121.841} C_VEL
LIN {X 0,Y 706.216,Z 977.729,A -85,B 0,C 180,E1 3123.502,E2 3123.502} C_VEL
LIN {X 0,Y 707.05,Z 981.016,A -85,B 0,C 180,E1 3124.357,E2 3124.357} C_VEL
LIN {X 0,Y 707.287,Z 981.346,A -85,B 0,C 180,E1 3124.636,E2 3124.636} C_VEL
LIN {X 0,Y 711.914,Z 995.199,A -85,B 0,C 180,E1 3124.963,E2 3124.963} C_VEL
LIN {X 0,Y 711.616,Z 1076.644,A -85,B 0,C 180,E1 3125.932,E2 3125.932} C_VEL
LIN {X 0,Y 711.04,Z 1117.464,A -85,B 0,C 180,E1 3126.935,E2 3126.935} C_VEL
LIN {X 0,Y 710.142,Z 1155.2,A -85,B 0,C 180,E1 3128.37,E2 3128.37} C_VEL
LIN {X 0,Y 709.204,Z 1190.369,A -85,B 0,C 180,E1 3130.239,E2 3130.239} C_VEL
LIN {X 0,Y 708.342,Z 1221.576,A -85,B 0,C 180,E1 3132.451,E2 3132.451} C_VEL
LIN {X 0,Y 707.662,Z 1248.479,A -85,B 0,C 180,E1 3134.93,E2 3134.93} C_VEL
LIN {X 0,Y 707.223,Z 1271.923,A -85,B 0,C 180,E1 3137.791,E2 3137.791} C_VEL
LIN {X 0,Y 706.917,Z 1290.2,A -85,B 0,C 180,E1 3140.826,E2 3140.826} C_VEL
LIN {X 0,Y 706.812,Z 1302.607,A -85,B 0,C 180,E1 3143.852,E2 3143.852} C_VEL
LIN {X 0,Y 706.794,Z 1308.959,A -85,B 0,C 180,E1 3146.318,E2 3146.318} C_VEL
LIN {X 0,Y 706.816,Z 1312.103,A -85,B 0,C 180,E1 3148.777,E2 3148.777} C_VEL
LIN {X 0,Y 706.793,Z 1312.094,A -85,B 0,C 180,E1 3151.234,E2 3151.234} C_VEL
LIN {X 0,Y 706.803,Z 1307.814,A -85,B 0,C 180,E1 3154.251,E2 3154.251} C_VEL
LIN {X 0,Y 706.969,Z 1296.926,A -85,B 0,C 180,E1 3157.704,E2 3157.704} C_VEL
LIN {X 0,Y 707.085,Z 1281.11,A -85,B 0,C 180,E1 3160.813,E2 3160.813} C_VEL
LIN {X 0,Y 707.491,Z 1259.832,A -85,B 0,C 180,E1 3163.79,E2 3163.79} C_VEL
LIN {X 0,Y 708.103,Z 1234.019,A -85,B 0,C 180,E1 3166.477,E2 3166.477} C_VEL
LIN {X 0,Y 708.861,Z 1203.985,A -85,B 0,C 180,E1 3168.869,E2 3168.869} C_VEL
LIN {X 0,Y 709.769,Z 1169.752,A -85,B 0,C 180,E1 3170.926,E2 3170.926} C_VEL
LIN {X 0,Y 710.719,Z 1132.11,A -85,B 0,C 180,E1 3172.573,E2 3172.573} C_VEL
LIN {X 0,Y 711.506,Z 1092.44,A -85,B 0,C 180,E1 3173.742,E2 3173.742} C_VEL
LIN {X 0,Y 711.886,Z 1052.802,A -85,B 0,C 180,E1 3174.41,E2 3174.41} C_VEL
LIN {X 0,Y 710.919,Z 990.882,A -85,B 0,C 180,E1 3175.121,E2 3175.121} C_VEL
LIN {X 0,Y 707.092,Z 981.007,A -85,B 0,C 180,E1 3175.384,E2 3175.384} C_VEL
LIN {X 0,Y 706.476,Z 979.552,A -85,B 0,C 180,E1 3176.221,E2 3176.221} C_VEL
LIN {X 0,Y 706.198,Z 977.53,A -85,B 0,C 180,E1 3176.649,E2 3176.649} C_VEL
LIN {X 0,Y 706.289,Z 977.53,A -85,B 0,C 180,E1 3180.997,E2 3180.997} C_VEL
LIN {X 0,Y 706.266,Z 977.53,A -85,B 0,C 180,E1 3185.41,E2 3185.41} C_VEL
LIN {X 0,Y 706.149,Z 977.53,A -85,B 0,C 180,E1 3190.079,E2 3190.079} C_VEL
LIN {X 0,Y 706.38,Z 977.53,A -85,B 0,C 180,E1 3195.071,E2 3195.071} C_VEL
LIN {X 0,Y 706.203,Z 977.53,A -85,B 0,C 180,E1 3200.582,E2 3200.582} C_VEL
LIN {X 0,Y 706.214,Z 977.53,A -85,B 0,C 180,E1 3206.107,E2 3206.107} C_VEL
LIN {X 0,Y 706.265,Z 977.53,A -85,B 0,C 180,E1 3210.446,E2 3210.446} C_VEL
LIN {X 0,Y 706.394,Z 977.53,A -85,B 0,C 180,E1 3214.608,E2 3214.608} C_VEL
LIN {X 0,Y 706.403,Z 977.53,A -85,B 0,C 180,E1 3218.626,E2 3218.626} C_VEL
LIN {X 0,Y 706.441,Z 977.53,A -85,B 0,C 180,E1 3223.82,E2 3223.82} C_VEL
LIN {X 0,Y 706.489,Z 977.53,A -85,B 0,C 180,E1 3228.881,E2 3228.881} C_VEL
LIN {X 0,Y 706.627,Z 977.53,A -85,B 0,C 180,E1 3233.855,E2 3233.855} C_VEL
LIN {X 0,Y 706.707,Z 977.53,A -85,B 0,C 180,E1 3236.821,E2 3236.821} C_VEL
LIN {X 0,Y 708.272,Z 995.48,A -85,B 0,C 180,E1 3237.058,E2 3237.058} C_VEL
LIN {X 0,Y 708.261,Z 1043.194,A -85,B 0,C 180,E1 3237.633,E2 3237.633} C_VEL
LIN {X 0,Y 707.952,Z 1071.536,A -85,B 0,C 180,E1 3238.438,E2 3238.438} C_VEL
LIN {X 0,Y 707.6,Z 1098.073,A -85,B 0,C 180,E1 3239.702,E2 3239.702} C_VEL
LIN {X 0,Y 707.328,Z 1119.563,A -85,B 0,C 180,E1 3241.236,E2 3241.236} C_VEL
LIN {X 0,Y 707.084,Z 1138.63,A -85,B 0,C 180,E1 3243.233,E2 3243.233} C_VEL
LIN {X 0,Y 706.961,Z 1151.188,A -85,B 0,C 180,E1 3245.235,E2 3245.235} C_VEL
LIN {X 0,Y 706.878,Z 1159.24,A -85,B 0,C 180,E1 3247.398,E2 3247.398} C_VEL
LIN {X 0,Y 706.858,Z 1162.411,A -85,B 0,C 180,E1 3249.882,E2 3249.882} C_VEL
LIN {X 0,Y 706.927,Z 1159.52,A -85,B 0,C 180,E1 3252.385,E2 3252.385} C_VEL
LIN {X 0,Y 706.966,Z 1151.561,A -85,B 0,C 180,E1 3254.594,E2 3254.594} C_VEL
LIN {X 0,Y 707.112,Z 1137.498,A -85,B 0,C 180,E1 3256.823,E2 3256.823} C_VEL
LIN {X 0,Y 707.354,Z 1118.627,A -85,B 0,C 180,E1 3258.75,E2 3258.75} C_VEL
LIN {X 0,Y 707.606,Z 1095.216,A -85,B 0,C 180,E1 3260.37,E2 3260.37} C_VEL
LIN {X 0,Y 707.967,Z 1069.269,A -85,B 0,C 180,E1 3261.558,E2 3261.558} C_VEL
LIN {X 0,Y 708.25,Z 1040.948,A -85,B 0,C 180,E1 3262.325,E2 3262.325} C_VEL
LIN {X 0,Y 707.449,Z 981.682,A -85,B 0,C 180,E1 3263.008,E2 3263.008} C_VEL
LIN {X 0,Y 706.685,Z 977.53,A -85,B 0,C 180,E1 3263.089,E2 3263.089} C_VEL
LIN {X 0,Y 706.285,Z 977.53,A -85,B 0,C 180,E1 3268.392,E2 3268.392} C_VEL
LIN {X 0,Y 706.264,Z 977.53,A -85,B 0,C 180,E1 3273.193,E2 3273.193} C_VEL
LIN {X 0,Y 706.254,Z 977.53,A -85,B 0,C 180,E1 3278.482,E2 3278.482} C_VEL
LIN {X 0,Y 706.431,Z 977.53,A -85,B 0,C 180,E1 3283.35,E2 3283.35} C_VEL
LIN {X 0,Y 706.155,Z 977.53,A -85,B 0,C 180,E1 3288.685,E2 3288.685} C_VEL
LIN {X 0,Y 706.153,Z 977.53,A -85,B 0,C 180,E1 3293.064,E2 3293.064} C_VEL
LIN {X 0,Y 706.243,Z 977.53,A -85,B 0,C 180,E1 3297.556,E2 3297.556} C_VEL
LIN {X 0,Y 706.275,Z 977.53,A -85,B 0,C 180,E1 3301.83,E2 3301.83} C_VEL
LIN {X 0,Y 706.394,Z 977.53,A -85,B 0,C 180,E1 3305.942,E2 3305.942} C_VEL
LIN {X 0,Y 706.409,Z 977.53,A -85,B 0,C 180,E1 3311.225,E2 3311.225} C_VEL
LIN {X 0,Y 706.352,Z 977.53,A -85,B 0,C 180,E1 3316.345,E2 3316.345} C_VEL
LIN {X 0,Y 706.516,Z 977.53,A -85,B 0,C 180,E1 3320.609,E2 3320.609} C_VEL
LIN {X 0,Y 706.529,Z 977.53,A -85,B 0,C 180,E1 3325.073,E2 3325.073} C_VEL
LIN {X 0,Y 706.582,Z 977.53,A -85,B 0,C 180,E1 3329.994,E2 3329.994} C_VEL
LIN {X 0,Y 706.723,Z 977.53,A -85,B 0,C 180,E1 3334.914,E2 3334.914} C_VEL
LIN {X 0,Y 706.446,Z 977.53,A -85,B 0,C 180,E1 3339.875,E2 3339.875} C_VEL
LIN {X 0,Y 706.439,Z 977.53,A -85,B 0,C 180,E1 3345.147,E2 3345.147} C_VEL
LIN {X 0,Y 706.449,Z 977.53,A -85,B 0,C 180,E1 3350.065,E2 3350.065} C_VEL
LIN {X 0,Y 706.325,Z 977.53,A -85,B 0,C 180,E1 3355.401,E2 3355.401} C_VEL
LIN {X 0,Y 706.282,Z 977.53,A -85,B 0,C 180,E1 3360.883,E2 3360.883} C_VEL
LIN {X 0,Y 706.299,Z 977.53,A -85,B 0,C 180,E1 3365.39,E2 3365.39} C_VEL
LIN {X 0,Y 706.156,Z 977.53,A -85,B 0,C 180,E1 3370.063,E2 3370.063} C_VEL
LIN {X 0,Y 706.372,Z 977.53,A -85,B 0,C 180,E1 3375.056,E2 3375.056} C_VEL
LIN {X 0,Y 706.226,Z 977.53,A -85,B 0,C 180,E1 3380.561,E2 3380.561} C_VEL
LIN {X 0,Y 706.216,Z 977.53,A -85,B 0,C 180,E1 3386.086,E2 3386.086} C_VEL
LIN {X 0,Y 706.272,Z 977.53,A -85,B 0,C 180,E1 3390.426,E2 3390.426} C_VEL
LIN {X 0,Y 706.545,Z 977.53,A -85,B 0,C 180,E1 3395.175,E2 3395.175} C_VEL
LIN {X 0,Y 711.748,Z 994.438,A -85,B 0,C 180,E1 3395.558,E2 3395.558} C_VEL
LIN {X 0,Y 711.492,Z 1036.019,A -85,B 0,C 180,E1 3396.301,E2 3396.301} C_VEL
LIN {X 0,Y 710.656,Z 1075.179,A -85,B 0,C 180,E1 3397.5,E2 3397.5} C_VEL
LIN {X 0,Y 709.723,Z 1111.438,A -85,B 0,C 180,E1 3399.121,E2 3399.121} C_VEL
LIN {X 0,Y 708.859,Z 1144.611,A -85,B 0,C 180,E1 3401.134,E2 3401.134} C_VEL
LIN {X 0,Y 708.041,Z 1174.52,A -85,B 0,C 180,E1 3403.52,E2 3403.52} C_VEL
LIN {X 0,Y 707.498,Z 1200.172,A -85,B 0,C 180,E1 3406.208,E2 3406.208} C_VEL
LIN {X 0,Y 707.089,Z 1221.389,A -85,B 0,C 180,E1 3409.185,E2 3409.185} C_VEL
LIN {X 0,Y 706.936,Z 1237.087,A -85,B 0,C 180,E1 3412.293,E2 3412.293} C_VEL
LIN {X 0,Y 706.843,Z 1246.265,A -85,B 0,C 180,E1 3415.073,E2 3415.073} C_VEL
LIN {X 0,Y 706.833,Z 1250.944,A -85,B 0,C 180,E1 3417.534,E2 3417.534} C_VEL
LIN {X 0,Y 706.787,Z 1252.497,A -85,B 0,C 180,E1 3419.991,E2 3419.991} C_VEL
LIN {X 0,Y 706.852,Z 1250.843,A -85,B 0,C 180,E1 3422.448,E2 3422.448} C_VEL
LIN {X 0,Y 706.89,Z 1244.408,A -85,B 0,C 180,E1 3425.526,E2 3425.526} C_VEL
LIN {X 0,Y 706.921,Z 1232.687,A -85,B 0,C 180,E1 3428.62,E2 3428.62} C_VEL
LIN {X 0,Y 707.19,Z 1214.933,A -85,B 0,C 180,E1 3431.734,E2 3431.734} C_VEL
LIN {X 0,Y 707.254,Z 1210.348,A -85,B 0,C 180,E1 3432.393,E2 3432.393} C_VEL
LIN {X 0,Y 703.509,Z 1201.764,A -85,B 0,C 180,E1 3433.599,E2 3433.599} C_VEL
LIN {X 0,Y 699.823,Z 1192.335,A -85,B 0,C 180,E1 3434.772,E2 3434.772} C_VEL
LIN {X 0,Y 700.609,Z 1164.597,A -85,B 0,C 180,E1 3437.451,E2 3437.451} C_VEL
LIN {X 0,Y 701.597,Z 1132.999,A -85,B 0,C 180,E1 3439.768,E2 3439.768} C_VEL
LIN {X 0,Y 702.625,Z 1098.066,A -85,B 0,C 180,E1 3441.691,E2 3441.691} C_VEL
LIN {X 0,Y 703.705,Z 1059.158,A -85,B 0,C 180,E1 3443.222,E2 3443.222} C_VEL
LIN {X 0,Y 704.408,Z 1018.726,A -85,B 0,C 180,E1 3444.245,E2 3444.245} C_VEL
LIN {X 0,Y 704.003,Z 993.448,A -85,B 0,C 180,E1 3444.65,E2 3444.65} C_VEL
LIN {X 0,Y 698.347,Z 977.53,A -85,B 0,C 180,E1 3445.071,E2 3445.071} C_VEL
LIN {X 0,Y 698.339,Z 977.53,A -85,B 0,C 180,E1 3449.923,E2 3449.923} C_VEL
LIN {X 0,Y 698.316,Z 977.53,A -85,B 0,C 180,E1 3454.467,E2 3454.467} C_VEL
LIN {X 0,Y 698.239,Z 977.53,A -85,B 0,C 180,E1 3458.984,E2 3458.984} C_VEL
LIN {X 0,Y 698.135,Z 977.53,A -85,B 0,C 180,E1 3464.263,E2 3464.263} C_VEL
LIN {X 0,Y 698.169,Z 977.53,A -85,B 0,C 180,E1 3469.409,E2 3469.409} C_VEL
LIN {X 0,Y 698.429,Z 977.53,A -85,B 0,C 180,E1 3474.15,E2 3474.15} C_VEL
LIN {X 0,Y 698.275,Z 977.53,A -85,B 0,C 180,E1 3478.621,E2 3478.621} C_VEL
LIN {X 0,Y 698.308,Z 977.925,A -85,B 0,C 180,E1 3482.475,E2 3482.475} C_VEL
LIN {X 0,Y 700.417,Z 982.901,A -85,B 0,C 180,E1 3482.986,E2 3482.986} C_VEL
LIN {X 0,Y 704.647,Z 988.507,A -85,B 0,C 180,E1 3484.263,E2 3484.263} C_VEL
LIN {X 0,Y 704.414,Z 994.627,A -85,B 0,C 180,E1 3484.672,E2 3484.672} C_VEL
LIN {X 0,Y 704.384,Z 1076.742,A -85,B 0,C 180,E1 3485.672,E2 3485.672} C_VEL
LIN {X 0,Y 703.726,Z 1118.028,A -85,B 0,C 180,E1 3486.699,E2 3486.699} C_VEL
LIN {X 0,Y 702.695,Z 1155.787,A -85,B 0,C 180,E1 3488.157,E2 3488.157} C_VEL
LIN {X 0,Y 701.594,Z 1192.239,A -85,B 0,C 180,E1 3490.136,E2 3490.136} C_VEL
LIN {X 0,Y 700.576,Z 1225.062,A -85,B 0,C 180,E1 3492.542,E2 3492.542} C_VEL
LIN {X 0,Y 699.78,Z 1251.681,A -85,B 0,C 180,E1 3495.106,E2 3495.106} C_VEL
LIN {X 0,Y 699.338,Z 1275.201,A -85,B 0,C 180,E1 3498.127,E2 3498.127} C_VEL
LIN {X 0,Y 698.99,Z 1292.864,A -85,B 0,C 180,E1 3501.278,E2 3501.278} C_VEL
LIN {X 0,Y 698.942,Z 1304.523,A -85,B 0,C 180,E1 3504.407,E2 3504.407} C_VEL
LIN {X 0,Y 698.875,Z 1310.927,A -85,B 0,C 180,E1 3507.52,E2 3507.52} C_VEL
LIN {X 0,Y 698.852,Z 1312.5,A -85,B 0,C 180,E1 3510.006,E2 3510.006} C_VEL
LIN {X 0,Y 698.887,Z 1310.911,A -85,B 0,C 180,E1 3512.491,E2 3512.491} C_VEL
LIN {X 0,Y 698.96,Z 1304.486,A -85,B 0,C 180,E1 3515.604,E2 3515.604} C_VEL
LIN {X 0,Y 698.993,Z 1292.813,A -85,B 0,C 180,E1 3518.734,E2 3518.734} C_VEL
LIN {X 0,Y 699.346,Z 1275.118,A -85,B 0,C 180,E1 3521.884,E2 3521.884} C_VEL
LIN {X 0,Y 699.805,Z 1251.573,A -85,B 0,C 180,E1 3524.905,E2 3524.905} C_VEL
LIN {X 0,Y 700.552,Z 1224.917,A -85,B 0,C 180,E1 3527.47,E2 3527.47} C_VEL
LIN {X 0,Y 701.596,Z 1192.234,A -85,B 0,C 180,E1 3529.865,E2 3529.865} C_VEL
LIN {X 0,Y 702.671,Z 1156.552,A -85,B 0,C 180,E1 3531.808,E2 3531.808} C_VEL
LIN {X 0,Y 703.751,Z 1117.768,A -85,B 0,C 180,E1 3533.308,E2 3533.308} C_VEL
LIN {X 0,Y 704.453,Z 1078.416,A -85,B 0,C 180,E1 3534.294,E2 3534.294} C_VEL
LIN {X 0,Y 704.637,Z 1007.358,A -85,B 0,C 180,E1 3535.179,E2 3535.179} C_VEL
LIN {X 0,Y 703.921,Z 993.041,A -85,B 0,C 180,E1 3535.385,E2 3535.385} C_VEL
LIN {X 0,Y 704.666,Z 988.435,A -85,B 0,C 180,E1 3535.739,E2 3535.739} C_VEL
LIN {X 0,Y 700.325,Z 982.801,A -85,B 0,C 180,E1 3537.031,E2 3537.031} C_VEL
LIN {X 0,Y 698.289,Z 977.53,A -85,B 0,C 180,E1 3537.573,E2 3537.573} C_VEL
LIN {X 0,Y 698.366,Z 977.53,A -85,B 0,C 180,E1 3542.856,E2 3542.856} C_VEL
LIN {X 0,Y 698.406,Z 977.53,A -85,B 0,C 180,E1 3547.415,E2 3547.415} C_VEL
LIN {X 0,Y 698.395,Z 977.53,A -85,B 0,C 180,E1 3552.487,E2 3552.487} C_VEL
LIN {X 0,Y 698.219,Z 977.53,A -85,B 0,C 180,E1 3557.738,E2 3557.738} C_VEL
